METHOD FB_init : BOOL
VAR_INPUT
	bInitRetains : BOOL; // if TRUE, the retain variables are initialized (warm start / cold start)
	bInCopyCode : BOOL;  // if TRUE, the instance afterwards gets moved into the copy code (online change)
END_VAR
AddInput('aElement', aElement);
AddInput('ipContainer', ipContainer);
AddInput('nIndex', nIndex);
AddInput('hrPrev', hrPrev);
AddOutput('ipContainer', ipContainer);
AddOutput('hresult',hresult);
END_METHOD

METHOD PUBLIC  Clone : I_Node
VAR
	pNode : POINTER TO Node_F_VN_SetAt_TcVnVector4_INT;
END_VAR
pNode := __NEW(Node_F_VN_SetAt_TcVnVector4_INT);
Clone := pNode^;
END_METHOD

METHOD PROTECTED OnExecute : HRESULT
hresult.Value := F_VN_SetAt_TcVnVector4_INT(
    aElement := aElement.Value,
    ipContainer := ipContainer.Value,
    nIndex := nIndex.Value,
    hrPrev:= hrPrev.Value);
END_METHOD

METHOD PUBLIC PreExecutionCheck
VAR_INPUT
	Check : I_PreExecutionChecks;
END_VAR
Check.IsTrue(ipContainer.IsValid, 'ipContainer must be a valid container');
END_METHOD

END_FUNCTION_BLOCK

// Nodes/Basic Container Operations/Node_F_VN_SetAt_TcVnVector4_LREAL
{attribute 'linkalways'} 
{attribute 'no_explicit_call' := 'This FB is a CLASS and must be accessed using methods or properties'}
{attribute 'enable_dynamic_creation'}
FUNCTION_BLOCK Node_F_VN_SetAt_TcVnVector4_LREAL EXTENDS VisionNode
VAR
    aElement : _TcVnVector4_LREAL;
    ipContainer : _ITcVnContainer;
    nIndex : _ULINT(0);
    hrPrev : _HRESULT(S_OK);
    hresult : _HRESULT(S_OK);
END_VAR

METHOD FB_init : BOOL
VAR_INPUT
	bInitRetains : BOOL; // if TRUE, the retain variables are initialized (warm start / cold start)
	bInCopyCode : BOOL;  // if TRUE, the instance afterwards gets moved into the copy code (online change)
END_VAR
AddInput('aElement', aElement);
AddInput('ipContainer', ipContainer);
AddInput('nIndex', nIndex);
AddInput('hrPrev', hrPrev);
AddOutput('ipContainer', ipContainer);
AddOutput('hresult',hresult);
END_METHOD

METHOD PUBLIC  Clone : I_Node
VAR
	pNode : POINTER TO Node_F_VN_SetAt_TcVnVector4_LREAL;
END_VAR
pNode := __NEW(Node_F_VN_SetAt_TcVnVector4_LREAL);
Clone := pNode^;
END_METHOD

METHOD PROTECTED OnExecute : HRESULT
hresult.Value := F_VN_SetAt_TcVnVector4_LREAL(
    aElement := aElement.Value,
    ipContainer := ipContainer.Value,
    nIndex := nIndex.Value,
    hrPrev:= hrPrev.Value);
END_METHOD

METHOD PUBLIC PreExecutionCheck
VAR_INPUT
	Check : I_PreExecutionChecks;
END_VAR
Check.IsTrue(ipContainer.IsValid, 'ipContainer must be a valid container');
END_METHOD

END_FUNCTION_BLOCK

// Nodes/Basic Container Operations/Node_F_VN_SetAt_TcVnVector4_SINT
{attribute 'linkalways'} 
{attribute 'no_explicit_call' := 'This FB is a CLASS and must be accessed using methods or properties'}
{attribute 'enable_dynamic_creation'}
FUNCTION_BLOCK Node_F_VN_SetAt_TcVnVector4_SINT EXTENDS VisionNode
VAR
    aElement : _TcVnVector4_SINT;
    ipContainer : _ITcVnContainer;
    nIndex : _ULINT(0);
    hrPrev : _HRESULT(S_OK);
    hresult : _HRESULT(S_OK);
END_VAR

METHOD FB_init : BOOL
VAR_INPUT
	bInitRetains : BOOL; // if TRUE, the retain variables are initialized (warm start / cold start)
	bInCopyCode : BOOL;  // if TRUE, the instance afterwards gets moved into the copy code (online change)
END_VAR
AddInput('aElement', aElement);
AddInput('ipContainer', ipContainer);
AddInput('nIndex', nIndex);
AddInput('hrPrev', hrPrev);
AddOutput('ipContainer', ipContainer);
AddOutput('hresult',hresult);
END_METHOD

METHOD PUBLIC  Clone : I_Node
VAR
	pNode : POINTER TO Node_F_VN_SetAt_TcVnVector4_SINT;
END_VAR
pNode := __NEW(Node_F_VN_SetAt_TcVnVector4_SINT);
Clone := pNode^;
END_METHOD

METHOD PROTECTED OnExecute : HRESULT
hresult.Value := F_VN_SetAt_TcVnVector4_SINT(
    aElement := aElement.Value,
    ipContainer := ipContainer.Value,
    nIndex := nIndex.Value,
    hrPrev:= hrPrev.Value);
END_METHOD

METHOD PUBLIC PreExecutionCheck
VAR_INPUT
	Check : I_PreExecutionChecks;
END_VAR
Check.IsTrue(ipContainer.IsValid, 'ipContainer must be a valid container');
END_METHOD

END_FUNCTION_BLOCK

// Nodes/Basic Container Operations/Node_F_VN_SetAt_TcVnVector4_UINT
{attribute 'linkalways'} 
{attribute 'no_explicit_call' := 'This FB is a CLASS and must be accessed using methods or properties'}
{attribute 'enable_dynamic_creation'}
FUNCTION_BLOCK Node_F_VN_SetAt_TcVnVector4_UINT EXTENDS VisionNode
VAR
    aElement : _TcVnVector4_UINT;
    ipContainer : _ITcVnContainer;
    nIndex : _ULINT(0);
    hrPrev : _HRESULT(S_OK);
    hresult : _HRESULT(S_OK);
END_VAR

METHOD FB_init : BOOL
VAR_INPUT
	bInitRetains : BOOL; // if TRUE, the retain variables are initialized (warm start / cold start)
	bInCopyCode : BOOL;  // if TRUE, the instance afterwards gets moved into the copy code (online change)
END_VAR
AddInput('aElement', aElement);
AddInput('ipContainer', ipContainer);
AddInput('nIndex', nIndex);
AddInput('hrPrev', hrPrev);
AddOutput('ipContainer', ipContainer);
AddOutput('hresult',hresult);
END_METHOD

METHOD PUBLIC  Clone : I_Node
VAR
	pNode : POINTER TO Node_F_VN_SetAt_TcVnVector4_UINT;
END_VAR
pNode := __NEW(Node_F_VN_SetAt_TcVnVector4_UINT);
Clone := pNode^;
END_METHOD

METHOD PROTECTED OnExecute : HRESULT
hresult.Value := F_VN_SetAt_TcVnVector4_UINT(
    aElement := aElement.Value,
    ipContainer := ipContainer.Value,
    nIndex := nIndex.Value,
    hrPrev:= hrPrev.Value);
END_METHOD

METHOD PUBLIC PreExecutionCheck
VAR_INPUT
	Check : I_PreExecutionChecks;
END_VAR
Check.IsTrue(ipContainer.IsValid, 'ipContainer must be a valid container');
END_METHOD

END_FUNCTION_BLOCK

// Nodes/Basic Container Operations/Node_F_VN_SetAt_TcVnVector4_USINT
{attribute 'linkalways'} 
{attribute 'no_explicit_call' := 'This FB is a CLASS and must be accessed using methods or properties'}
{attribute 'enable_dynamic_creation'}
FUNCTION_BLOCK Node_F_VN_SetAt_TcVnVector4_USINT EXTENDS VisionNode
VAR
    aElement : _TcVnVector4_USINT;
    ipContainer : _ITcVnContainer;
    nIndex : _ULINT(0);
    hrPrev : _HRESULT(S_OK);
    hresult : _HRESULT(S_OK);
END_VAR

METHOD FB_init : BOOL
VAR_INPUT
	bInitRetains : BOOL; // if TRUE, the retain variables are initialized (warm start / cold start)
	bInCopyCode : BOOL;  // if TRUE, the instance afterwards gets moved into the copy code (online change)
END_VAR
AddInput('aElement', aElement);
AddInput('ipContainer', ipContainer);
AddInput('nIndex', nIndex);
AddInput('hrPrev', hrPrev);
AddOutput('ipContainer', ipContainer);
AddOutput('hresult',hresult);
END_METHOD

METHOD PUBLIC  Clone : I_Node
VAR
	pNode : POINTER TO Node_F_VN_SetAt_TcVnVector4_USINT;
END_VAR
pNode := __NEW(Node_F_VN_SetAt_TcVnVector4_USINT);
Clone := pNode^;
END_METHOD

METHOD PROTECTED OnExecute : HRESULT
hresult.Value := F_VN_SetAt_TcVnVector4_USINT(
    aElement := aElement.Value,
    ipContainer := ipContainer.Value,
    nIndex := nIndex.Value,
    hrPrev:= hrPrev.Value);
END_METHOD

METHOD PUBLIC PreExecutionCheck
VAR_INPUT
	Check : I_PreExecutionChecks;
END_VAR
Check.IsTrue(ipContainer.IsValid, 'ipContainer must be a valid container');
END_METHOD

END_FUNCTION_BLOCK

// Nodes/Basic Container Operations/Node_F_VN_SetAt_UDINT
{attribute 'linkalways'} 
{attribute 'no_explicit_call' := 'This FB is a CLASS and must be accessed using methods or properties'}
{attribute 'enable_dynamic_creation'}
FUNCTION_BLOCK Node_F_VN_SetAt_UDINT EXTENDS VisionNode
VAR
    nElement : _UDINT(0);
    ipContainer : _ITcVnContainer;
    nIndex : _ULINT(0);
    hrPrev : _HRESULT(S_OK);
    hresult : _HRESULT(S_OK);
END_VAR

METHOD FB_init : BOOL
VAR_INPUT
	bInitRetains : BOOL; // if TRUE, the retain variables are initialized (warm start / cold start)
	bInCopyCode : BOOL;  // if TRUE, the instance afterwards gets moved into the copy code (online change)
END_VAR
AddInput('nElement', nElement);
AddInput('ipContainer', ipContainer);
AddInput('nIndex', nIndex);
AddInput('hrPrev', hrPrev);
AddOutput('ipContainer', ipContainer);
AddOutput('hresult',hresult);
END_METHOD

METHOD PUBLIC  Clone : I_Node
VAR
	pNode : POINTER TO Node_F_VN_SetAt_UDINT;
END_VAR
pNode := __NEW(Node_F_VN_SetAt_UDINT);
Clone := pNode^;
END_METHOD

METHOD PROTECTED OnExecute : HRESULT
hresult.Value := F_VN_SetAt_UDINT(
    nElement := nElement.Value,
    ipContainer := ipContainer.Value,
    nIndex := nIndex.Value,
    hrPrev:= hrPrev.Value);
END_METHOD

METHOD PUBLIC PreExecutionCheck
VAR_INPUT
	Check : I_PreExecutionChecks;
END_VAR
Check.IsTrue(ipContainer.IsValid, 'ipContainer must be a valid container');
Check.IsTrue(ipContainer.HasType('CTcVnContainer_Vector_UDINT'), 'ipContainer contains incorrect types');
END_METHOD

END_FUNCTION_BLOCK

// Nodes/Basic Container Operations/Node_F_VN_SetAt_UINT
{attribute 'linkalways'} 
{attribute 'no_explicit_call' := 'This FB is a CLASS and must be accessed using methods or properties'}
{attribute 'enable_dynamic_creation'}
FUNCTION_BLOCK Node_F_VN_SetAt_UINT EXTENDS VisionNode
VAR
    nElement : _UINT(0);
    ipContainer : _ITcVnContainer;
    nIndex : _ULINT(0);
    hrPrev : _HRESULT(S_OK);
    hresult : _HRESULT(S_OK);
END_VAR

METHOD FB_init : BOOL
VAR_INPUT
	bInitRetains : BOOL; // if TRUE, the retain variables are initialized (warm start / cold start)
	bInCopyCode : BOOL;  // if TRUE, the instance afterwards gets moved into the copy code (online change)
END_VAR
AddInput('nElement', nElement);
AddInput('ipContainer', ipContainer);
AddInput('nIndex', nIndex);
AddInput('hrPrev', hrPrev);
AddOutput('ipContainer', ipContainer);
AddOutput('hresult',hresult);
END_METHOD

METHOD PUBLIC  Clone : I_Node
VAR
	pNode : POINTER TO Node_F_VN_SetAt_UINT;
END_VAR
pNode := __NEW(Node_F_VN_SetAt_UINT);
Clone := pNode^;
END_METHOD

METHOD PROTECTED OnExecute : HRESULT
hresult.Value := F_VN_SetAt_UINT(
    nElement := nElement.Value,
    ipContainer := ipContainer.Value,
    nIndex := nIndex.Value,
    hrPrev:= hrPrev.Value);
END_METHOD

METHOD PUBLIC PreExecutionCheck
VAR_INPUT
	Check : I_PreExecutionChecks;
END_VAR
Check.IsTrue(ipContainer.IsValid, 'ipContainer must be a valid container');
Check.IsTrue(ipContainer.HasType('CTcVnContainer_Vector_UINT'), 'ipContainer contains incorrect types');
END_METHOD

END_FUNCTION_BLOCK

// Nodes/Basic Container Operations/Node_F_VN_SetAt_ULINT
{attribute 'linkalways'} 
{attribute 'no_explicit_call' := 'This FB is a CLASS and must be accessed using methods or properties'}
{attribute 'enable_dynamic_creation'}
FUNCTION_BLOCK Node_F_VN_SetAt_ULINT EXTENDS VisionNode
VAR
    nElement : _ULINT(0);
    ipContainer : _ITcVnContainer;
    nIndex : _ULINT(0);
    hrPrev : _HRESULT(S_OK);
    hresult : _HRESULT(S_OK);
END_VAR

METHOD FB_init : BOOL
VAR_INPUT
	bInitRetains : BOOL; // if TRUE, the retain variables are initialized (warm start / cold start)
	bInCopyCode : BOOL;  // if TRUE, the instance afterwards gets moved into the copy code (online change)
END_VAR
AddInput('nElement', nElement);
AddInput('ipContainer', ipContainer);
AddInput('nIndex', nIndex);
AddInput('hrPrev', hrPrev);
AddOutput('ipContainer', ipContainer);
AddOutput('hresult',hresult);
END_METHOD

METHOD PUBLIC  Clone : I_Node
VAR
	pNode : POINTER TO Node_F_VN_SetAt_ULINT;
END_VAR
pNode := __NEW(Node_F_VN_SetAt_ULINT);
Clone := pNode^;
END_METHOD

METHOD PROTECTED OnExecute : HRESULT
hresult.Value := F_VN_SetAt_ULINT(
    nElement := nElement.Value,
    ipContainer := ipContainer.Value,
    nIndex := nIndex.Value,
    hrPrev:= hrPrev.Value);
END_METHOD

METHOD PUBLIC PreExecutionCheck
VAR_INPUT
	Check : I_PreExecutionChecks;
END_VAR
Check.IsTrue(ipContainer.IsValid, 'ipContainer must be a valid container');
Check.IsTrue(ipContainer.HasType('CTcVnContainer_Vector_ULINT'), 'ipContainer contains incorrect types');
END_METHOD

END_FUNCTION_BLOCK

// Nodes/Basic Container Operations/Node_F_VN_SetAt_USINT
{attribute 'linkalways'} 
{attribute 'no_explicit_call' := 'This FB is a CLASS and must be accessed using methods or properties'}
{attribute 'enable_dynamic_creation'}
FUNCTION_BLOCK Node_F_VN_SetAt_USINT EXTENDS VisionNode
VAR
    nElement : _USINT(0);
    ipContainer : _ITcVnContainer;
    nIndex : _ULINT(0);
    hrPrev : _HRESULT(S_OK);
    hresult : _HRESULT(S_OK);
END_VAR

METHOD FB_init : BOOL
VAR_INPUT
	bInitRetains : BOOL; // if TRUE, the retain variables are initialized (warm start / cold start)
	bInCopyCode : BOOL;  // if TRUE, the instance afterwards gets moved into the copy code (online change)
END_VAR
AddInput('nElement', nElement);
AddInput('ipContainer', ipContainer);
AddInput('nIndex', nIndex);
AddInput('hrPrev', hrPrev);
AddOutput('ipContainer', ipContainer);
AddOutput('hresult',hresult);
END_METHOD

METHOD PUBLIC  Clone : I_Node
VAR
	pNode : POINTER TO Node_F_VN_SetAt_USINT;
END_VAR
pNode := __NEW(Node_F_VN_SetAt_USINT);
Clone := pNode^;
END_METHOD

METHOD PROTECTED OnExecute : HRESULT
hresult.Value := F_VN_SetAt_USINT(
    nElement := nElement.Value,
    ipContainer := ipContainer.Value,
    nIndex := nIndex.Value,
    hrPrev:= hrPrev.Value);
END_METHOD

METHOD PUBLIC PreExecutionCheck
VAR_INPUT
	Check : I_PreExecutionChecks;
END_VAR
Check.IsTrue(ipContainer.IsValid, 'ipContainer must be a valid container');
Check.IsTrue(ipContainer.HasType('CTcVnContainer_Vector_USINT'), 'ipContainer contains incorrect types');
END_METHOD

END_FUNCTION_BLOCK

// Nodes/Basic Image Operations/Node_F_VN_CopyImage
{attribute 'linkalways'} 
{attribute 'no_explicit_call' := 'This FB is a CLASS and must be accessed using methods or properties'}
{attribute 'enable_dynamic_creation'}
FUNCTION_BLOCK Node_F_VN_CopyImage EXTENDS VisionNode
VAR
    ipSrcImage : _ITcVnImage;
    ipDestImage : _ITcVnImage;
    hrPrev : _HRESULT(S_OK);
	hresult : _HRESULT(S_OK);
END_VAR

METHOD FB_init : BOOL
VAR_INPUT
	bInitRetains : BOOL; // if TRUE, the retain variables are initialized (warm start / cold start)
	bInCopyCode : BOOL;  // if TRUE, the instance afterwards gets moved into the copy code (online change)
END_VAR
AddInput('ipSrcImage', ipSrcImage);
AddInput('hrPrev', hrPrev);
AddOutput('ipDestImage', ipDestImage);
AddOutput('hresult',hresult);
END_METHOD

METHOD PUBLIC  Clone : I_Node
VAR
	pNode : POINTER TO Node_F_VN_CopyImage;
END_VAR
pNode := __NEW(Node_F_VN_CopyImage);
Clone := pNode^;
END_METHOD

METHOD PROTECTED OnExecute : HRESULT
hresult.Value := F_VN_CopyImage(
    ipSrcImage := ipSrcImage.Value,
	ipDestImage := ipDestImage.Value,
	hrPrev:= hrPrev.Value);
END_METHOD

METHOD PUBLIC PreExecutionCheck
VAR_INPUT
	Check : I_PreExecutionChecks;
END_VAR
Check.IsTrue(ipSrcImage.IsValid, 'ipSrcImage must contain an image');
END_METHOD

END_FUNCTION_BLOCK

// Nodes/Basic Image Operations/Node_F_VN_GetImageChannel
{attribute 'linkalways'} 
{attribute 'no_explicit_call' := 'This FB is a CLASS and must be accessed using methods or properties'}
{attribute 'enable_dynamic_creation'}
FUNCTION_BLOCK Node_F_VN_GetImageChannel EXTENDS VisionNode
VAR
    ipSrcImage : _ITcVnImage;
    ipDestImage : _ITcVnImage;
    nChannelIndex : _UINT(0);
    hrPrev : _HRESULT(S_OK);
	hresult : _HRESULT(S_OK);
END_VAR

METHOD FB_init : BOOL
VAR_INPUT
	bInitRetains : BOOL; // if TRUE, the retain variables are initialized (warm start / cold start)
	bInCopyCode : BOOL;  // if TRUE, the instance afterwards gets moved into the copy code (online change)
END_VAR
AddInput('ipSrcImage', ipSrcImage);
AddInput('hrPrev', hrPrev);
AddOutput('ipDestImage', ipDestImage);
AddOutput('hresult',hresult);
AddParameter('nChannelIndex', nChannelIndex);
END_METHOD

METHOD PUBLIC  Clone : I_Node
VAR
	pNode : POINTER TO Node_F_VN_GetImageChannel;
END_VAR
pNode := __NEW(Node_F_VN_GetImageChannel);
Clone := pNode^;
END_METHOD

METHOD PROTECTED OnExecute : HRESULT
hresult.Value := F_VN_GetImageChannel(
    ipSrcImage := ipSrcImage.Value,
	ipDestImage := ipDestImage.Value,
    nChannelIndex := nChannelIndex.Value,
	hrPrev:= hrPrev.Value);
END_METHOD

METHOD PUBLIC PreExecutionCheck
VAR_INPUT
	Check : I_PreExecutionChecks;
END_VAR
Check.IsTrue(ipSrcImage.IsValid, 'ipSrcImage must contain an image');
END_METHOD

END_FUNCTION_BLOCK

// Nodes/Basic Image Operations/Node_F_VN_GetImageHeight
{attribute 'linkalways'} 
{attribute 'no_explicit_call' := 'This FB is a CLASS and must be accessed using methods or properties'}
{attribute 'enable_dynamic_creation'}
FUNCTION_BLOCK Node_F_VN_GetImageHeight EXTENDS VisionNode
VAR
    ipImage : _ITcVnImage;
    nHeight : _UDINT(0);
    hrPrev : _HRESULT(S_OK);
	hresult : _HRESULT(S_OK);
END_VAR

METHOD FB_init : BOOL
VAR_INPUT
	bInitRetains : BOOL; // if TRUE, the retain variables are initialized (warm start / cold start)
	bInCopyCode : BOOL;  // if TRUE, the instance afterwards gets moved into the copy code (online change)
END_VAR
AddInput('ipImage', ipImage);
AddInput('hrPrev', hrPrev);
AddOutput('nHeight', nHeight);
AddOutput('hresult', hresult);
END_METHOD

METHOD PUBLIC  Clone : I_Node
VAR
	pNode : POINTER TO Node_F_VN_GetImageHeight;
END_VAR
pNode := __NEW(Node_F_VN_GetImageHeight);
Clone := pNode^;
END_METHOD

METHOD PROTECTED OnExecute : HRESULT
hresult.Value := F_VN_GetImageHeight(
    ipImage := ipImage.Value,
    nHeight := nHeight.Value,
	hrPrev:= hrPrev.Value);
END_METHOD

METHOD PUBLIC PreExecutionCheck
VAR_INPUT
	Check : I_PreExecutionChecks;
END_VAR
Check.IsTrue(ipImage.IsValid, 'ipImage must contain an image');
END_METHOD

END_FUNCTION_BLOCK

// Nodes/Basic Image Operations/Node_F_VN_GetImageInfo
{attribute 'linkalways'} 
{attribute 'no_explicit_call' := 'This FB is a CLASS and must be accessed using methods or properties'}
{attribute 'enable_dynamic_creation'}
FUNCTION_BLOCK Node_F_VN_GetImageInfo EXTENDS VisionNode
VAR
    ipImage : _ITcVnImage;
    stImageInfo : _TcVnImageInfo;
    hrPrev : _HRESULT(S_OK);
	hresult : _HRESULT(S_OK);
END_VAR

METHOD FB_init : BOOL
VAR_INPUT
	bInitRetains : BOOL; // if TRUE, the retain variables are initialized (warm start / cold start)
	bInCopyCode : BOOL;  // if TRUE, the instance afterwards gets moved into the copy code (online change)
END_VAR
AddInput('ipImage', ipImage);
AddInput('hrPrev', hrPrev);
AddOutput('stImageInfo', stImageInfo);
AddOutput('hresult',hresult);
END_METHOD

METHOD PUBLIC  Clone : I_Node
VAR
	pNode : POINTER TO Node_F_VN_GetImageInfo;
END_VAR
pNode := __NEW(Node_F_VN_GetImageInfo);
Clone := pNode^;
END_METHOD

METHOD PROTECTED OnExecute : HRESULT
hresult.Value := F_VN_GetImageInfo(
    ipImage := ipImage.Value,
	stImageInfo := stImageInfo.Value,
	hrPrev:= hrPrev.Value);
END_METHOD

METHOD PUBLIC PreExecutionCheck
VAR_INPUT
	Check : I_PreExecutionChecks;
END_VAR
Check.IsTrue(ipImage.IsValid, 'ipImage must contain an image');
END_METHOD

END_FUNCTION_BLOCK

// Nodes/Basic Image Operations/Node_F_VN_GetImageWidth
{attribute 'linkalways'} 
{attribute 'no_explicit_call' := 'This FB is a CLASS and must be accessed using methods or properties'}
{attribute 'enable_dynamic_creation'}
FUNCTION_BLOCK Node_F_VN_GetImageWidth EXTENDS VisionNode
VAR
    ipImage : _ITcVnImage;
    nWidth : _UDINT(0);
    hrPrev : _HRESULT(S_OK);
	hresult : _HRESULT(S_OK);
END_VAR

METHOD FB_init : BOOL
VAR_INPUT
	bInitRetains : BOOL; // if TRUE, the retain variables are initialized (warm start / cold start)
	bInCopyCode : BOOL;  // if TRUE, the instance afterwards gets moved into the copy code (online change)
END_VAR
AddInput('ipImage', ipImage);
AddInput('hrPrev', hrPrev);
AddOutput('nWidth', nWidth);
AddOutput('hresult',hresult);
END_METHOD

METHOD PUBLIC  Clone : I_Node
VAR
	pNode : POINTER TO Node_F_VN_GetImageWidth;
END_VAR
pNode := __NEW(Node_F_VN_GetImageWidth);
Clone := pNode^;
END_METHOD

METHOD PROTECTED OnExecute : HRESULT
hresult.Value := F_VN_GetImageWidth(
    ipImage := ipImage.Value,
    nWidth := nWidth.Value,
	hrPrev:= hrPrev.Value);
END_METHOD

METHOD PUBLIC PreExecutionCheck
VAR_INPUT
	Check : I_PreExecutionChecks;
END_VAR
Check.IsTrue(ipImage.IsValid, 'ipImage must contain an image');
END_METHOD

END_FUNCTION_BLOCK

// Nodes/Basic Image Operations/Node_F_VN_GetPixelFormat
{attribute 'linkalways'} 
{attribute 'no_explicit_call' := 'This FB is a CLASS and must be accessed using methods or properties'}
{attribute 'enable_dynamic_creation'}
FUNCTION_BLOCK Node_F_VN_GetPixelFormat EXTENDS VisionNode
VAR
    ipImage : _ITcVnImage;
    stPixelFormat : _TcVnPixelFormat;
    hrPrev : _HRESULT(S_OK);
	hresult : _HRESULT(S_OK);
END_VAR

METHOD FB_init : BOOL
VAR_INPUT
	bInitRetains : BOOL; // if TRUE, the retain variables are initialized (warm start / cold start)
	bInCopyCode : BOOL;  // if TRUE, the instance afterwards gets moved into the copy code (online change)
END_VAR
AddInput('ipImage', ipImage);
AddInput('hrPrev', hrPrev);
AddOutput('stPixelFormat', stPixelFormat);
AddOutput('hresult',hresult);
END_METHOD

METHOD PUBLIC  Clone : I_Node
VAR
	pNode : POINTER TO Node_F_VN_GetPixelFormat;
END_VAR
pNode := __NEW(Node_F_VN_GetPixelFormat);
Clone := pNode^;
END_METHOD

METHOD PROTECTED OnExecute : HRESULT
hresult.Value := F_VN_GetPixelFormat(
    ipImage := ipImage.Value,
	stPixelFormat := stPixelFormat.Value,
	hrPrev:= hrPrev.Value);
END_METHOD

METHOD PUBLIC PreExecutionCheck
VAR_INPUT
	Check : I_PreExecutionChecks;
END_VAR
Check.IsTrue(ipImage.IsValid, 'ipImage must contain an image');
END_METHOD

END_FUNCTION_BLOCK

// Nodes/Basic Image Operations/Node_F_VN_SetRoi
{attribute 'linkalways'} 
{attribute 'no_explicit_call' := 'This FB is a CLASS and must be accessed using methods or properties'}
{attribute 'enable_dynamic_creation'}
FUNCTION_BLOCK Node_F_VN_SetRoi EXTENDS VisionNode
VAR
    nX : _UDINT(0);
    nY : _UDINT(0);
    nWidth : _UDINT(0);
    nHeight : _UDINT(0);
    ipDestImage : _ITcVnImage;
    hrPrev : _HRESULT(S_OK);
	hresult : _HRESULT(S_OK);
END_VAR

METHOD FB_init : BOOL
VAR_INPUT
	bInitRetains : BOOL; // if TRUE, the retain variables are initialized (warm start / cold start)
	bInCopyCode : BOOL;  // if TRUE, the instance afterwards gets moved into the copy code (online change)
END_VAR
AddParameter('nX', nX);
AddParameter('nY', nY);
AddParameter('nWidth', nWidth);
AddParameter('nHeight', nHeight);
AddInput('ipDestImage', ipDestImage);
AddInput('hrPrev', hrPrev);
AddOutput('ipDestImage', ipDestImage);
AddOutput('hresult',hresult);
END_METHOD

METHOD PUBLIC  Clone : I_Node
VAR
	pNode : POINTER TO Node_F_VN_SetRoi;
END_VAR
pNode := __NEW(Node_F_VN_SetRoi);
Clone := pNode^;
END_METHOD

METHOD PROTECTED  OnExecute : HRESULT
hresult.Value := F_VN_SetRoi(
    nX := nX.Value,
    nY := nY.Value,
    nWidth := nWidth.Value,
	nHeight := nHeight.Value,
	ipDestImage := ipDestImage.Value,
	hrPrev:= hrPrev.Value);
END_METHOD

METHOD PUBLIC PreExecutionCheck
VAR_INPUT
	Check : I_PreExecutionChecks;
END_VAR
Check.IsTrue(ipDestImage.IsValid, 'ipDestImage must contain an image');
END_METHOD

END_FUNCTION_BLOCK

// Nodes/Constants/Node_RGBA_BLACK
{attribute 'linkalways'} 
{attribute 'no_explicit_call' := 'This FB is a CLASS and must be accessed using methods or properties'}
{attribute 'enable_dynamic_creation'}
FUNCTION_BLOCK Node_RGBA_BLACK EXTENDS VisionNode
VAR
    out : _TcVnVector4_LREAL;
END_VAR

METHOD FB_init : BOOL
VAR_INPUT
	bInitRetains : BOOL; // if TRUE, the retain variables are initialized (warm start / cold start)
	bInCopyCode : BOOL;  // if TRUE, the instance afterwards gets moved into the copy code (online change)
END_VAR
AddOutput('out', out);
END_METHOD

METHOD PUBLIC  Clone : I_Node
VAR
	pNode : POINTER TO Node_RGBA_BLACK;
END_VAR
pNode := __NEW(Node_RGBA_BLACK);
Clone := pNode^;
END_METHOD

METHOD PROTECTED OnExecute : HRESULT
out.Value := GVL_COLOURS.RGBA_BLACK;
END_METHOD

METHOD PUBLIC PreExecutionCheck
VAR_INPUT
	Check : I_PreExecutionChecks;
END_VAR
END_METHOD

END_FUNCTION_BLOCK

// Nodes/Constants/Node_RGBA_BLUE
{attribute 'linkalways'} 
{attribute 'no_explicit_call' := 'This FB is a CLASS and must be accessed using methods or properties'}
{attribute 'enable_dynamic_creation'}
FUNCTION_BLOCK Node_RGBA_BLUE EXTENDS VisionNode
VAR
    out : _TcVnVector4_LREAL;
END_VAR

METHOD FB_init : BOOL
VAR_INPUT
	bInitRetains : BOOL; // if TRUE, the retain variables are initialized (warm start / cold start)
	bInCopyCode : BOOL;  // if TRUE, the instance afterwards gets moved into the copy code (online change)
END_VAR
AddOutput('out', out);
END_METHOD

METHOD PUBLIC  Clone : I_Node
VAR
	pNode : POINTER TO Node_RGBA_BLUE;
END_VAR
pNode := __NEW(Node_RGBA_BLUE);
Clone := pNode^;
END_METHOD

METHOD PROTECTED OnExecute : HRESULT
out.Value := GVL_COLOURS.RGBA_BLUE;
END_METHOD

METHOD PUBLIC PreExecutionCheck
VAR_INPUT
	Check : I_PreExecutionChecks;
END_VAR
END_METHOD

END_FUNCTION_BLOCK

// Nodes/Constants/Node_RGBA_CYAN
{attribute 'linkalways'} 
{attribute 'no_explicit_call' := 'This FB is a CLASS and must be accessed using methods or properties'}
{attribute 'enable_dynamic_creation'}
FUNCTION_BLOCK Node_RGBA_CYAN EXTENDS VisionNode
VAR
    out : _TcVnVector4_LREAL;
END_VAR

METHOD FB_init : BOOL
VAR_INPUT
	bInitRetains : BOOL; // if TRUE, the retain variables are initialized (warm start / cold start)
	bInCopyCode : BOOL;  // if TRUE, the instance afterwards gets moved into the copy code (online change)
END_VAR
AddOutput('out', out);
END_METHOD

METHOD PUBLIC  Clone : I_Node
VAR
	pNode : POINTER TO Node_RGBA_CYAN;
END_VAR
pNode := __NEW(Node_RGBA_CYAN);
Clone := pNode^;
END_METHOD

METHOD PROTECTED OnExecute : HRESULT
out.Value := GVL_COLOURS.RGBA_CYAN;
END_METHOD

METHOD PUBLIC PreExecutionCheck
VAR_INPUT
	Check : I_PreExecutionChecks;
END_VAR
END_METHOD

END_FUNCTION_BLOCK

// Nodes/Constants/Node_RGBA_GREEN
{attribute 'linkalways'} 
{attribute 'no_explicit_call' := 'This FB is a CLASS and must be accessed using methods or properties'}
{attribute 'enable_dynamic_creation'}
FUNCTION_BLOCK Node_RGBA_GREEN EXTENDS VisionNode
VAR
    out : _TcVnVector4_LREAL;
END_VAR

METHOD FB_init : BOOL
VAR_INPUT
	bInitRetains : BOOL; // if TRUE, the retain variables are initialized (warm start / cold start)
	bInCopyCode : BOOL;  // if TRUE, the instance afterwards gets moved into the copy code (online change)
END_VAR
AddOutput('out', out);
END_METHOD

METHOD PUBLIC  Clone : I_Node
VAR
	pNode : POINTER TO Node_RGBA_GREEN;
END_VAR
pNode := __NEW(Node_RGBA_GREEN);
Clone := pNode^;
END_METHOD

METHOD PROTECTED OnExecute : HRESULT
out.Value := GVL_COLOURS.RGBA_GREEN;
END_METHOD

METHOD PUBLIC PreExecutionCheck
VAR_INPUT
	Check : I_PreExecutionChecks;
END_VAR
END_METHOD

END_FUNCTION_BLOCK

// Nodes/Constants/Node_RGBA_MAGENTA
{attribute 'linkalways'} 
{attribute 'no_explicit_call' := 'This FB is a CLASS and must be accessed using methods or properties'}
{attribute 'enable_dynamic_creation'}
FUNCTION_BLOCK Node_RGBA_MAGENTA EXTENDS VisionNode
VAR
    out : _TcVnVector4_LREAL;
END_VAR

METHOD FB_init : BOOL
VAR_INPUT
	bInitRetains : BOOL; // if TRUE, the retain variables are initialized (warm start / cold start)
	bInCopyCode : BOOL;  // if TRUE, the instance afterwards gets moved into the copy code (online change)
END_VAR
AddOutput('out', out);
END_METHOD

METHOD PUBLIC  Clone : I_Node
VAR
	pNode : POINTER TO Node_RGBA_MAGENTA;
END_VAR
pNode := __NEW(Node_RGBA_MAGENTA);
Clone := pNode^;
END_METHOD

METHOD PROTECTED OnExecute : HRESULT
out.Value := GVL_COLOURS.RGBA_MAGENTA;
END_METHOD

METHOD PUBLIC PreExecutionCheck
VAR_INPUT
	Check : I_PreExecutionChecks;
END_VAR
END_METHOD

END_FUNCTION_BLOCK

// Nodes/Constants/Node_RGBA_RED
{attribute 'linkalways'} 
{attribute 'no_explicit_call' := 'This FB is a CLASS and must be accessed using methods or properties'}
{attribute 'enable_dynamic_creation'}
FUNCTION_BLOCK Node_RGBA_RED EXTENDS VisionNode
VAR
    out : _TcVnVector4_LREAL;
END_VAR

METHOD FB_init : BOOL
VAR_INPUT
	bInitRetains : BOOL; // if TRUE, the retain variables are initialized (warm start / cold start)
	bInCopyCode : BOOL;  // if TRUE, the instance afterwards gets moved into the copy code (online change)
END_VAR
AddOutput('out', out);
END_METHOD

METHOD PUBLIC  Clone : I_Node
VAR
	pNode : POINTER TO Node_RGBA_RED;
END_VAR
pNode := __NEW(Node_RGBA_RED);
Clone := pNode^;
END_METHOD

METHOD PROTECTED OnExecute : HRESULT
out.Value := GVL_COLOURS.RGBA_RED;
END_METHOD

METHOD PUBLIC PreExecutionCheck
VAR_INPUT
	Check : I_PreExecutionChecks;
END_VAR
END_METHOD

END_FUNCTION_BLOCK

// Nodes/Constants/Node_RGBA_WHITE
{attribute 'linkalways'} 
{attribute 'no_explicit_call' := 'This FB is a CLASS and must be accessed using methods or properties'}
{attribute 'enable_dynamic_creation'}
FUNCTION_BLOCK Node_RGBA_WHITE EXTENDS VisionNode
VAR
    out : _TcVnVector4_LREAL;
END_VAR

METHOD FB_init : BOOL
VAR_INPUT
	bInitRetains : BOOL; // if TRUE, the retain variables are initialized (warm start / cold start)
	bInCopyCode : BOOL;  // if TRUE, the instance afterwards gets moved into the copy code (online change)
END_VAR
AddOutput('out', out);
END_METHOD

METHOD PUBLIC  Clone : I_Node
VAR
	pNode : POINTER TO Node_RGBA_WHITE;
END_VAR
pNode := __NEW(Node_RGBA_WHITE);
Clone := pNode^;
END_METHOD

METHOD PROTECTED OnExecute : HRESULT
out.Value := GVL_COLOURS.RGBA_WHITE;
END_METHOD

METHOD PUBLIC PreExecutionCheck
VAR_INPUT
	Check : I_PreExecutionChecks;
END_VAR
END_METHOD

END_FUNCTION_BLOCK

// Nodes/Constants/Node_RGBA_YELLOW
{attribute 'linkalways'} 
{attribute 'no_explicit_call' := 'This FB is a CLASS and must be accessed using methods or properties'}
{attribute 'enable_dynamic_creation'}
FUNCTION_BLOCK Node_RGBA_YELLOW EXTENDS VisionNode
VAR
    out : _TcVnVector4_LREAL;
END_VAR

METHOD FB_init : BOOL
VAR_INPUT
	bInitRetains : BOOL; // if TRUE, the retain variables are initialized (warm start / cold start)
	bInCopyCode : BOOL;  // if TRUE, the instance afterwards gets moved into the copy code (online change)
END_VAR
AddOutput('out', out);
END_METHOD

METHOD PUBLIC  Clone : I_Node
VAR
	pNode : POINTER TO Node_RGBA_YELLOW;
END_VAR
pNode := __NEW(Node_RGBA_YELLOW);
Clone := pNode^;
END_METHOD

METHOD PROTECTED OnExecute : HRESULT
out.Value := GVL_COLOURS.RGBA_YELLOW;
END_METHOD

METHOD PUBLIC PreExecutionCheck
VAR_INPUT
	Check : I_PreExecutionChecks;
END_VAR
END_METHOD

END_FUNCTION_BLOCK

// Nodes/Container Statistics/Node_F_VN_MaxElementElementwise_DINT
{attribute 'linkalways'} 
{attribute 'no_explicit_call' := 'This FB is a CLASS and must be accessed using methods or properties'}
{attribute 'enable_dynamic_creation'}
FUNCTION_BLOCK Node_F_VN_MaxElementElementwise_DINT EXTENDS VisionNode
VAR
    ipContainer : _ITcVnContainer;
    nMax : _DINT(0);
    hrPrev : _HRESULT(S_OK);
    hresult : _HRESULT(S_OK);
END_VAR

METHOD FB_init : BOOL
VAR_INPUT
	bInitRetains : BOOL; // if TRUE, the retain variables are initialized (warm start / cold start)
	bInCopyCode : BOOL;  // if TRUE, the instance afterwards gets moved into the copy code (online change)
END_VAR
AddInput('ipContainer', ipContainer);
AddInput('nMax', nMax);
AddInput('hrPrev', hrPrev);
AddOutput('ipContainer', ipContainer);
AddOutput('hresult',hresult);
END_METHOD

METHOD PUBLIC  Clone : I_Node
VAR
	pNode : POINTER TO Node_F_VN_MaxElementElementwise_DINT;
END_VAR
pNode := __NEW(Node_F_VN_MaxElementElementwise_DINT);
Clone := pNode^;
END_METHOD

METHOD PROTECTED OnExecute : HRESULT
hresult.Value := F_VN_MaxElementElementwise_DINT(
    ipContainer := ipContainer.Value,
    nMax := nMax.Value,
    hrPrev:= hrPrev.Value);
END_METHOD

METHOD PUBLIC PreExecutionCheck
VAR_INPUT
	Check : I_PreExecutionChecks;
END_VAR
VAR
    name : STRING;
END_VAR
Check.IsTrue(ipContainer.IsValid, 'ipContainer must be a valid container');
Check.IsTrue(ipContainer.HasType('CTcVnContainer_Vector_DINT'), 'ipContainer contains incorrect types');
END_METHOD

END_FUNCTION_BLOCK

// Nodes/Container Statistics/Node_F_VN_MaxElementElementwise_INT
{attribute 'linkalways'} 
{attribute 'no_explicit_call' := 'This FB is a CLASS and must be accessed using methods or properties'}
{attribute 'enable_dynamic_creation'}
FUNCTION_BLOCK Node_F_VN_MaxElementElementwise_INT EXTENDS VisionNode
VAR
    ipContainer : _ITcVnContainer;
    nMax : _INT(0);
    hrPrev : _HRESULT(S_OK);
    hresult : _HRESULT(S_OK);
END_VAR

METHOD FB_init : BOOL
VAR_INPUT
	bInitRetains : BOOL; // if TRUE, the retain variables are initialized (warm start / cold start)
	bInCopyCode : BOOL;  // if TRUE, the instance afterwards gets moved into the copy code (online change)
END_VAR
AddInput('ipContainer', ipContainer);
AddInput('nMax', nMax);
AddInput('hrPrev', hrPrev);
AddOutput('ipContainer', ipContainer);
AddOutput('hresult',hresult);
END_METHOD

METHOD PUBLIC  Clone : I_Node
VAR
	pNode : POINTER TO Node_F_VN_MaxElementElementwise_INT;
END_VAR
pNode := __NEW(Node_F_VN_MaxElementElementwise_INT);
Clone := pNode^;
END_METHOD

METHOD PROTECTED OnExecute : HRESULT
hresult.Value := F_VN_MaxElementElementwise_INT(
    ipContainer := ipContainer.Value,
    nMax := nMax.Value,
    hrPrev:= hrPrev.Value);
END_METHOD

METHOD PUBLIC PreExecutionCheck
VAR_INPUT
	Check : I_PreExecutionChecks;
END_VAR
Check.IsTrue(ipContainer.IsValid, 'ipContainer must be a valid container');
Check.IsTrue(ipContainer.HasType('CTcVnContainer_Vector_INT'), 'ipContainer contains incorrect types');
END_METHOD

END_FUNCTION_BLOCK

// Nodes/Container Statistics/Node_F_VN_MaxElementElementwise_LREAL
{attribute 'linkalways'} 
{attribute 'no_explicit_call' := 'This FB is a CLASS and must be accessed using methods or properties'}
{attribute 'enable_dynamic_creation'}
FUNCTION_BLOCK Node_F_VN_MaxElementElementwise_LREAL EXTENDS VisionNode
VAR
    ipContainer : _ITcVnContainer;
    fMax : _LREAL(0.0);
    hrPrev : _HRESULT(S_OK);
    hresult : _HRESULT(S_OK);
END_VAR

METHOD FB_init : BOOL
VAR_INPUT
	bInitRetains : BOOL; // if TRUE, the retain variables are initialized (warm start / cold start)
	bInCopyCode : BOOL;  // if TRUE, the instance afterwards gets moved into the copy code (online change)
END_VAR
AddInput('ipContainer', ipContainer);
AddInput('fMax', fMax);
AddInput('hrPrev', hrPrev);
AddOutput('ipContainer', ipContainer);
AddOutput('hresult',hresult);
END_METHOD

METHOD PUBLIC  Clone : I_Node
VAR
	pNode : POINTER TO Node_F_VN_MaxElementElementwise_LREAL;
END_VAR
pNode := __NEW(Node_F_VN_MaxElementElementwise_LREAL);
Clone := pNode^;
END_METHOD

METHOD PROTECTED OnExecute : HRESULT
hresult.Value := F_VN_MaxElementElementwise_LREAL(
    ipContainer := ipContainer.Value,
    fMax := fMax.Value,
    hrPrev:= hrPrev.Value);
END_METHOD

METHOD PUBLIC PreExecutionCheck
VAR_INPUT
	Check : I_PreExecutionChecks;
END_VAR
Check.IsTrue(ipContainer.IsValid, 'ipContainer must be a valid container');
Check.IsTrue(ipContainer.HasType('CTcVnContainer_Vector_LREAL'), 'ipContainer contains incorrect types');
END_METHOD

END_FUNCTION_BLOCK

// Nodes/Container Statistics/Node_F_VN_MaxElementElementwise_REAL
{attribute 'linkalways'} 
{attribute 'no_explicit_call' := 'This FB is a CLASS and must be accessed using methods or properties'}
{attribute 'enable_dynamic_creation'}
FUNCTION_BLOCK Node_F_VN_MaxElementElementwise_REAL EXTENDS VisionNode
VAR
    ipContainer : _ITcVnContainer;
    fMax : _REAL(0.0);
    hrPrev : _HRESULT(S_OK);
    hresult : _HRESULT(S_OK);
END_VAR

METHOD FB_init : BOOL
VAR_INPUT
	bInitRetains : BOOL; // if TRUE, the retain variables are initialized (warm start / cold start)
	bInCopyCode : BOOL;  // if TRUE, the instance afterwards gets moved into the copy code (online change)
END_VAR
AddInput('ipContainer', ipContainer);
AddInput('fMax', fMax);
AddInput('hrPrev', hrPrev);
AddOutput('ipContainer', ipContainer);
AddOutput('hresult',hresult);
END_METHOD

METHOD PUBLIC  Clone : I_Node
VAR
	pNode : POINTER TO Node_F_VN_MaxElementElementwise_REAL;
END_VAR
pNode := __NEW(Node_F_VN_MaxElementElementwise_REAL);
Clone := pNode^;
END_METHOD

METHOD PROTECTED OnExecute : HRESULT
hresult.Value := F_VN_MaxElementElementwise_REAL(
    ipContainer := ipContainer.Value,
    fMax := fMax.Value,
    hrPrev:= hrPrev.Value);
END_METHOD

METHOD PUBLIC PreExecutionCheck
VAR_INPUT
	Check : I_PreExecutionChecks;
END_VAR
Check.IsTrue(ipContainer.IsValid, 'ipContainer must be a valid container');
Check.IsTrue(ipContainer.HasType('CTcVnContainer_Vector_REAL'), 'ipContainer contains incorrect types');
END_METHOD

END_FUNCTION_BLOCK

// Nodes/Container Statistics/Node_F_VN_MaxElementElementwise_SINT
{attribute 'linkalways'} 
{attribute 'no_explicit_call' := 'This FB is a CLASS and must be accessed using methods or properties'}
{attribute 'enable_dynamic_creation'}
FUNCTION_BLOCK Node_F_VN_MaxElementElementwise_SINT EXTENDS VisionNode
VAR
    ipContainer : _ITcVnContainer;
    nMax : _SINT(0);
    hrPrev : _HRESULT(S_OK);
    hresult : _HRESULT(S_OK);
END_VAR

METHOD FB_init : BOOL
VAR_INPUT
	bInitRetains : BOOL; // if TRUE, the retain variables are initialized (warm start / cold start)
	bInCopyCode : BOOL;  // if TRUE, the instance afterwards gets moved into the copy code (online change)
END_VAR
AddInput('ipContainer', ipContainer);
AddInput('nMax', nMax);
AddInput('hrPrev', hrPrev);
AddOutput('ipContainer', ipContainer);
AddOutput('hresult',hresult);
END_METHOD

METHOD PUBLIC  Clone : I_Node
VAR
	pNode : POINTER TO Node_F_VN_MaxElementElementwise_SINT;
END_VAR
pNode := __NEW(Node_F_VN_MaxElementElementwise_SINT);
Clone := pNode^;
END_METHOD

METHOD PROTECTED OnExecute : HRESULT
hresult.Value := F_VN_MaxElementElementwise_SINT(
    ipContainer := ipContainer.Value,
    nMax := nMax.Value,
    hrPrev:= hrPrev.Value);
END_METHOD

METHOD PUBLIC PreExecutionCheck
VAR_INPUT
	Check : I_PreExecutionChecks;
END_VAR
Check.IsTrue(ipContainer.IsValid, 'ipContainer must be a valid container');
Check.IsTrue(ipContainer.HasType('CTcVnContainer_Vector_SINT'), 'ipContainer contains incorrect types');
END_METHOD

END_FUNCTION_BLOCK

// Nodes/Container Statistics/Node_F_VN_MaxElementElementwise_TcVnPoint2_DINT
{attribute 'linkalways'} 
{attribute 'no_explicit_call' := 'This FB is a CLASS and must be accessed using methods or properties'}
{attribute 'enable_dynamic_creation'}
FUNCTION_BLOCK Node_F_VN_MaxElementElementwise_TcVnPoint2_DINT EXTENDS VisionNode
VAR
    ipContainer : _ITcVnContainer;
    aMax : _TcVnPoint2_DINT;
    hrPrev : _HRESULT(S_OK);
    hresult : _HRESULT(S_OK);
END_VAR

METHOD FB_init : BOOL
VAR_INPUT
	bInitRetains : BOOL; // if TRUE, the retain variables are initialized (warm start / cold start)
	bInCopyCode : BOOL;  // if TRUE, the instance afterwards gets moved into the copy code (online change)
END_VAR
AddInput('ipContainer', ipContainer);
AddInput('aMax', aMax);
AddInput('hrPrev', hrPrev);
AddOutput('ipContainer', ipContainer);
AddOutput('hresult',hresult);
END_METHOD

METHOD PUBLIC  Clone : I_Node
VAR
	pNode : POINTER TO Node_F_VN_MaxElementElementwise_TcVnPoint2_DINT;
END_VAR
pNode := __NEW(Node_F_VN_MaxElementElementwise_TcVnPoint2_DINT);
Clone := pNode^;
END_METHOD

METHOD PROTECTED OnExecute : HRESULT
hresult.Value := F_VN_MaxElementElementwise_TcVnPoint2_DINT(
    ipContainer := ipContainer.Value,
    aMax := aMax.Value,
    hrPrev:= hrPrev.Value);
END_METHOD

METHOD PUBLIC PreExecutionCheck
VAR_INPUT
	Check : I_PreExecutionChecks;
END_VAR
Check.IsTrue(ipContainer.IsValid, 'ipContainer must be a valid container');
END_METHOD

END_FUNCTION_BLOCK

// Nodes/Container Statistics/Node_F_VN_MaxElementElementwise_TcVnPoint2_LREAL
{attribute 'linkalways'} 
{attribute 'no_explicit_call' := 'This FB is a CLASS and must be accessed using methods or properties'}
{attribute 'enable_dynamic_creation'}
FUNCTION_BLOCK Node_F_VN_MaxElementElementwise_TcVnPoint2_LREAL EXTENDS VisionNode
VAR
    ipContainer : _ITcVnContainer;
    aMax : _TcVnPoint2_LREAL;
    hrPrev : _HRESULT(S_OK);
    hresult : _HRESULT(S_OK);
END_VAR

METHOD FB_init : BOOL
VAR_INPUT
	bInitRetains : BOOL; // if TRUE, the retain variables are initialized (warm start / cold start)
	bInCopyCode : BOOL;  // if TRUE, the instance afterwards gets moved into the copy code (online change)
END_VAR
AddInput('ipContainer', ipContainer);
AddInput('aMax', aMax);
AddInput('hrPrev', hrPrev);
AddOutput('ipContainer', ipContainer);
AddOutput('hresult',hresult);
END_METHOD

METHOD PUBLIC  Clone : I_Node
VAR
	pNode : POINTER TO Node_F_VN_MaxElementElementwise_TcVnPoint2_LREAL;
END_VAR
pNode := __NEW(Node_F_VN_MaxElementElementwise_TcVnPoint2_LREAL);
Clone := pNode^;
END_METHOD

METHOD PROTECTED OnExecute : HRESULT
hresult.Value := F_VN_MaxElementElementwise_TcVnPoint2_LREAL(
    ipContainer := ipContainer.Value,
    aMax := aMax.Value,
    hrPrev:= hrPrev.Value);
END_METHOD

METHOD PUBLIC PreExecutionCheck
VAR_INPUT
	Check : I_PreExecutionChecks;
END_VAR
Check.IsTrue(ipContainer.IsValid, 'ipContainer must be a valid container');
END_METHOD

END_FUNCTION_BLOCK

// Nodes/Container Statistics/Node_F_VN_MaxElementElementwise_TcVnPoint2_REAL
{attribute 'linkalways'} 
{attribute 'no_explicit_call' := 'This FB is a CLASS and must be accessed using methods or properties'}
{attribute 'enable_dynamic_creation'}
FUNCTION_BLOCK Node_F_VN_MaxElementElementwise_TcVnPoint2_REAL EXTENDS VisionNode
VAR
    ipContainer : _ITcVnContainer;
    aMax : _TcVnPoint2_REAL;
    hrPrev : _HRESULT(S_OK);
    hresult : _HRESULT(S_OK);
END_VAR

METHOD FB_init : BOOL
VAR_INPUT
	bInitRetains : BOOL; // if TRUE, the retain variables are initialized (warm start / cold start)
	bInCopyCode : BOOL;  // if TRUE, the instance afterwards gets moved into the copy code (online change)
END_VAR
AddInput('ipContainer', ipContainer);
AddInput('aMax', aMax);
AddInput('hrPrev', hrPrev);
AddOutput('ipContainer', ipContainer);
AddOutput('hresult',hresult);
END_METHOD

METHOD PUBLIC  Clone : I_Node
VAR
	pNode : POINTER TO Node_F_VN_MaxElementElementwise_TcVnPoint2_REAL;
END_VAR
pNode := __NEW(Node_F_VN_MaxElementElementwise_TcVnPoint2_REAL);
Clone := pNode^;
END_METHOD

METHOD PROTECTED OnExecute : HRESULT
hresult.Value := F_VN_MaxElementElementwise_TcVnPoint2_REAL(
    ipContainer := ipContainer.Value,
    aMax := aMax.Value,
    hrPrev:= hrPrev.Value);
END_METHOD

METHOD PUBLIC PreExecutionCheck
VAR_INPUT
	Check : I_PreExecutionChecks;
END_VAR
Check.IsTrue(ipContainer.IsValid, 'ipContainer must be a valid container');
END_METHOD

END_FUNCTION_BLOCK

// Nodes/Container Statistics/Node_F_VN_MaxElementElementwise_TcVnPoint3_LREAL
{attribute 'linkalways'} 
{attribute 'no_explicit_call' := 'This FB is a CLASS and must be accessed using methods or properties'}
{attribute 'enable_dynamic_creation'}
FUNCTION_BLOCK Node_F_VN_MaxElementElementwise_TcVnPoint3_LREAL EXTENDS VisionNode
VAR
    ipContainer : _ITcVnContainer;
    aMax : _TcVnPoint3_LREAL;
    hrPrev : _HRESULT(S_OK);
    hresult : _HRESULT(S_OK);
END_VAR

METHOD FB_init : BOOL
VAR_INPUT
	bInitRetains : BOOL; // if TRUE, the retain variables are initialized (warm start / cold start)
	bInCopyCode : BOOL;  // if TRUE, the instance afterwards gets moved into the copy code (online change)
END_VAR
AddInput('ipContainer', ipContainer);
AddInput('aMax', aMax);
AddInput('hrPrev', hrPrev);
AddOutput('ipContainer', ipContainer);
AddOutput('hresult',hresult);
END_METHOD

METHOD PUBLIC  Clone : I_Node
VAR
	pNode : POINTER TO Node_F_VN_MaxElementElementwise_TcVnPoint3_LREAL;
END_VAR
pNode := __NEW(Node_F_VN_MaxElementElementwise_TcVnPoint3_LREAL);
Clone := pNode^;
END_METHOD

METHOD PROTECTED OnExecute : HRESULT
hresult.Value := F_VN_MaxElementElementwise_TcVnPoint3_LREAL(
    ipContainer := ipContainer.Value,
    aMax := aMax.Value,
    hrPrev:= hrPrev.Value);
END_METHOD

METHOD PUBLIC PreExecutionCheck
VAR_INPUT
	Check : I_PreExecutionChecks;
END_VAR
Check.IsTrue(ipContainer.IsValid, 'ipContainer must be a valid container');
END_METHOD

END_FUNCTION_BLOCK

// Nodes/Container Statistics/Node_F_VN_MaxElementElementwise_TcVnPoint3_REAL
{attribute 'linkalways'} 
{attribute 'no_explicit_call' := 'This FB is a CLASS and must be accessed using methods or properties'}
{attribute 'enable_dynamic_creation'}
FUNCTION_BLOCK Node_F_VN_MaxElementElementwise_TcVnPoint3_REAL EXTENDS VisionNode
VAR
    ipContainer : _ITcVnContainer;
    aMax : _TcVnPoint3_REAL;
    hrPrev : _HRESULT(S_OK);
    hresult : _HRESULT(S_OK);
END_VAR

METHOD FB_init : BOOL
VAR_INPUT
	bInitRetains : BOOL; // if TRUE, the retain variables are initialized (warm start / cold start)
	bInCopyCode : BOOL;  // if TRUE, the instance afterwards gets moved into the copy code (online change)
END_VAR
AddInput('ipContainer', ipContainer);
AddInput('aMax', aMax);
AddInput('hrPrev', hrPrev);
AddOutput('ipContainer', ipContainer);
AddOutput('hresult',hresult);
END_METHOD

METHOD PUBLIC  Clone : I_Node
VAR
	pNode : POINTER TO Node_F_VN_MaxElementElementwise_TcVnPoint3_REAL;
END_VAR
pNode := __NEW(Node_F_VN_MaxElementElementwise_TcVnPoint3_REAL);
Clone := pNode^;
END_METHOD

METHOD PROTECTED OnExecute : HRESULT
hresult.Value := F_VN_MaxElementElementwise_TcVnPoint3_REAL(
    ipContainer := ipContainer.Value,
    aMax := aMax.Value,
    hrPrev:= hrPrev.Value);
END_METHOD

METHOD PUBLIC PreExecutionCheck
VAR_INPUT
	Check : I_PreExecutionChecks;
END_VAR
Check.IsTrue(ipContainer.IsValid, 'ipContainer must be a valid container');
END_METHOD

END_FUNCTION_BLOCK

// Nodes/Container Statistics/Node_F_VN_MaxElementElementwise_TcVnVector2_DINT
{attribute 'linkalways'} 
{attribute 'no_explicit_call' := 'This FB is a CLASS and must be accessed using methods or properties'}
{attribute 'enable_dynamic_creation'}
FUNCTION_BLOCK Node_F_VN_MaxElementElementwise_TcVnVector2_DINT EXTENDS VisionNode
VAR
    ipContainer : _ITcVnContainer;
    aMax : _TcVnVector2_DINT;
    hrPrev : _HRESULT(S_OK);
    hresult : _HRESULT(S_OK);
END_VAR

METHOD FB_init : BOOL
VAR_INPUT
	bInitRetains : BOOL; // if TRUE, the retain variables are initialized (warm start / cold start)
	bInCopyCode : BOOL;  // if TRUE, the instance afterwards gets moved into the copy code (online change)
END_VAR
AddInput('ipContainer', ipContainer);
AddInput('aMax', aMax);
AddInput('hrPrev', hrPrev);
AddOutput('ipContainer', ipContainer);
AddOutput('hresult',hresult);
END_METHOD

METHOD PUBLIC  Clone : I_Node
VAR
	pNode : POINTER TO Node_F_VN_MaxElementElementwise_TcVnVector2_DINT;
END_VAR
pNode := __NEW(Node_F_VN_MaxElementElementwise_TcVnVector2_DINT);
Clone := pNode^;
END_METHOD

METHOD PROTECTED OnExecute : HRESULT
hresult.Value := F_VN_MaxElementElementwise_TcVnVector2_DINT(
    ipContainer := ipContainer.Value,
    aMax := aMax.Value,
    hrPrev:= hrPrev.Value);
END_METHOD

METHOD PUBLIC PreExecutionCheck
VAR_INPUT
	Check : I_PreExecutionChecks;
END_VAR
Check.IsTrue(ipContainer.IsValid, 'ipContainer must be a valid container');
END_METHOD

END_FUNCTION_BLOCK

// Nodes/Container Statistics/Node_F_VN_MaxElementElementwise_TcVnVector2_INT
{attribute 'linkalways'} 
{attribute 'no_explicit_call' := 'This FB is a CLASS and must be accessed using methods or properties'}
{attribute 'enable_dynamic_creation'}
FUNCTION_BLOCK Node_F_VN_MaxElementElementwise_TcVnVector2_INT EXTENDS VisionNode
VAR
    ipContainer : _ITcVnContainer;
    aMax : _TcVnVector2_INT;
    hrPrev : _HRESULT(S_OK);
    hresult : _HRESULT(S_OK);
END_VAR

METHOD FB_init : BOOL
VAR_INPUT
	bInitRetains : BOOL; // if TRUE, the retain variables are initialized (warm start / cold start)
	bInCopyCode : BOOL;  // if TRUE, the instance afterwards gets moved into the copy code (online change)
END_VAR
AddInput('ipContainer', ipContainer);
AddInput('aMax', aMax);
AddInput('hrPrev', hrPrev);
AddOutput('ipContainer', ipContainer);
AddOutput('hresult',hresult);
END_METHOD

METHOD PUBLIC  Clone : I_Node
VAR
	pNode : POINTER TO Node_F_VN_MaxElementElementwise_TcVnVector2_INT;
END_VAR
pNode := __NEW(Node_F_VN_MaxElementElementwise_TcVnVector2_INT);
Clone := pNode^;
END_METHOD

METHOD PROTECTED OnExecute : HRESULT
hresult.Value := F_VN_MaxElementElementwise_TcVnVector2_INT(
    ipContainer := ipContainer.Value,
    aMax := aMax.Value,
    hrPrev:= hrPrev.Value);
END_METHOD

METHOD PUBLIC PreExecutionCheck
VAR_INPUT
	Check : I_PreExecutionChecks;
END_VAR
Check.IsTrue(ipContainer.IsValid, 'ipContainer must be a valid container');
END_METHOD

END_FUNCTION_BLOCK

// Nodes/Container Statistics/Node_F_VN_MaxElementElementwise_TcVnVector2_REAL
{attribute 'linkalways'} 
{attribute 'no_explicit_call' := 'This FB is a CLASS and must be accessed using methods or properties'}
{attribute 'enable_dynamic_creation'}
FUNCTION_BLOCK Node_F_VN_MaxElementElementwise_TcVnVector2_REAL EXTENDS VisionNode
VAR
    ipContainer : _ITcVnContainer;
    aMax : _TcVnVector2_REAL;
    hrPrev : _HRESULT(S_OK);
    hresult : _HRESULT(S_OK);
END_VAR

METHOD FB_init : BOOL
VAR_INPUT
	bInitRetains : BOOL; // if TRUE, the retain variables are initialized (warm start / cold start)
	bInCopyCode : BOOL;  // if TRUE, the instance afterwards gets moved into the copy code (online change)
END_VAR
AddInput('ipContainer', ipContainer);
AddInput('aMax', aMax);
AddInput('hrPrev', hrPrev);
AddOutput('ipContainer', ipContainer);
AddOutput('hresult',hresult);
END_METHOD

METHOD PUBLIC  Clone : I_Node
VAR
	pNode : POINTER TO Node_F_VN_MaxElementElementwise_TcVnVector2_REAL;
END_VAR
pNode := __NEW(Node_F_VN_MaxElementElementwise_TcVnVector2_REAL);
Clone := pNode^;
END_METHOD

METHOD PROTECTED OnExecute : HRESULT
hresult.Value := F_VN_MaxElementElementwise_TcVnVector2_REAL(
    ipContainer := ipContainer.Value,
    aMax := aMax.Value,
    hrPrev:= hrPrev.Value);
END_METHOD

METHOD PUBLIC PreExecutionCheck
VAR_INPUT
	Check : I_PreExecutionChecks;
END_VAR
Check.IsTrue(ipContainer.IsValid, 'ipContainer must be a valid container');
END_METHOD

END_FUNCTION_BLOCK

// Nodes/Container Statistics/Node_F_VN_MaxElementElementwise_TcVnVector2_SINT
{attribute 'linkalways'} 
{attribute 'no_explicit_call' := 'This FB is a CLASS and must be accessed using methods or properties'}
{attribute 'enable_dynamic_creation'}
FUNCTION_BLOCK Node_F_VN_MaxElementElementwise_TcVnVector2_SINT EXTENDS VisionNode
VAR
    ipContainer : _ITcVnContainer;
    aMax : _TcVnVector2_SINT;
    hrPrev : _HRESULT(S_OK);
    hresult : _HRESULT(S_OK);
END_VAR

METHOD FB_init : BOOL
VAR_INPUT
	bInitRetains : BOOL; // if TRUE, the retain variables are initialized (warm start / cold start)
	bInCopyCode : BOOL;  // if TRUE, the instance afterwards gets moved into the copy code (online change)
END_VAR
AddInput('ipContainer', ipContainer);
AddInput('aMax', aMax);
AddInput('hrPrev', hrPrev);
AddOutput('ipContainer', ipContainer);
AddOutput('hresult',hresult);
END_METHOD

METHOD PUBLIC  Clone : I_Node
VAR
	pNode : POINTER TO Node_F_VN_MaxElementElementwise_TcVnVector2_SINT;
END_VAR
pNode := __NEW(Node_F_VN_MaxElementElementwise_TcVnVector2_SINT);
Clone := pNode^;
END_METHOD

METHOD PROTECTED OnExecute : HRESULT
hresult.Value := F_VN_MaxElementElementwise_TcVnVector2_SINT(
    ipContainer := ipContainer.Value,
    aMax := aMax.Value,
    hrPrev:= hrPrev.Value);
END_METHOD

METHOD PUBLIC PreExecutionCheck
VAR_INPUT
	Check : I_PreExecutionChecks;
END_VAR
Check.IsTrue(ipContainer.IsValid, 'ipContainer must be a valid container');
END_METHOD

END_FUNCTION_BLOCK

// Nodes/Container Statistics/Node_F_VN_MaxElementElementwise_TcVnVector2_UINT
{attribute 'linkalways'} 
{attribute 'no_explicit_call' := 'This FB is a CLASS and must be accessed using methods or properties'}
{attribute 'enable_dynamic_creation'}
FUNCTION_BLOCK Node_F_VN_MaxElementElementwise_TcVnVector2_UINT EXTENDS VisionNode
VAR
    ipContainer : _ITcVnContainer;
    aMax : _TcVnVector2_UINT;
    hrPrev : _HRESULT(S_OK);
    hresult : _HRESULT(S_OK);
END_VAR

METHOD FB_init : BOOL
VAR_INPUT
	bInitRetains : BOOL; // if TRUE, the retain variables are initialized (warm start / cold start)
	bInCopyCode : BOOL;  // if TRUE, the instance afterwards gets moved into the copy code (online change)
END_VAR
AddInput('ipContainer', ipContainer);
AddInput('aMax', aMax);
AddInput('hrPrev', hrPrev);
AddOutput('ipContainer', ipContainer);
AddOutput('hresult',hresult);
END_METHOD

METHOD PUBLIC  Clone : I_Node
VAR
	pNode : POINTER TO Node_F_VN_MaxElementElementwise_TcVnVector2_UINT;
END_VAR
pNode := __NEW(Node_F_VN_MaxElementElementwise_TcVnVector2_UINT);
Clone := pNode^;
END_METHOD

METHOD PROTECTED OnExecute : HRESULT
hresult.Value := F_VN_MaxElementElementwise_TcVnVector2_UINT(
    ipContainer := ipContainer.Value,
    aMax := aMax.Value,
    hrPrev:= hrPrev.Value);
END_METHOD

METHOD PUBLIC PreExecutionCheck
VAR_INPUT
	Check : I_PreExecutionChecks;
END_VAR
Check.IsTrue(ipContainer.IsValid, 'ipContainer must be a valid container');
END_METHOD

END_FUNCTION_BLOCK

// Nodes/Container Statistics/Node_F_VN_MaxElementElementwise_TcVnVector2_USINT
{attribute 'linkalways'} 
{attribute 'no_explicit_call' := 'This FB is a CLASS and must be accessed using methods or properties'}
{attribute 'enable_dynamic_creation'}
FUNCTION_BLOCK Node_F_VN_MaxElementElementwise_TcVnVector2_USINT EXTENDS VisionNode
VAR
    ipContainer : _ITcVnContainer;
    aMax : _TcVnVector2_USINT;
    hrPrev : _HRESULT(S_OK);
    hresult : _HRESULT(S_OK);
END_VAR

METHOD FB_init : BOOL
VAR_INPUT
	bInitRetains : BOOL; // if TRUE, the retain variables are initialized (warm start / cold start)
	bInCopyCode : BOOL;  // if TRUE, the instance afterwards gets moved into the copy code (online change)
END_VAR
AddInput('ipContainer', ipContainer);
AddInput('aMax', aMax);
AddInput('hrPrev', hrPrev);
AddOutput('ipContainer', ipContainer);
AddOutput('hresult',hresult);
END_METHOD

METHOD PUBLIC  Clone : I_Node
VAR
	pNode : POINTER TO Node_F_VN_MaxElementElementwise_TcVnVector2_USINT;
END_VAR
pNode := __NEW(Node_F_VN_MaxElementElementwise_TcVnVector2_USINT);
Clone := pNode^;
END_METHOD

METHOD PROTECTED OnExecute : HRESULT
hresult.Value := F_VN_MaxElementElementwise_TcVnVector2_USINT(
    ipContainer := ipContainer.Value,
    aMax := aMax.Value,
    hrPrev:= hrPrev.Value);
END_METHOD

METHOD PUBLIC PreExecutionCheck
VAR_INPUT
	Check : I_PreExecutionChecks;
END_VAR
Check.IsTrue(ipContainer.IsValid, 'ipContainer must be a valid container');
END_METHOD

END_FUNCTION_BLOCK

// Nodes/Container Statistics/Node_F_VN_MaxElementElementwise_TcVnVector3_INT
{attribute 'linkalways'} 
{attribute 'no_explicit_call' := 'This FB is a CLASS and must be accessed using methods or properties'}
{attribute 'enable_dynamic_creation'}
FUNCTION_BLOCK Node_F_VN_MaxElementElementwise_TcVnVector3_INT EXTENDS VisionNode
VAR
    ipContainer : _ITcVnContainer;
    aMax : _TcVnVector3_INT;
    hrPrev : _HRESULT(S_OK);
    hresult : _HRESULT(S_OK);
END_VAR

METHOD FB_init : BOOL
VAR_INPUT
	bInitRetains : BOOL; // if TRUE, the retain variables are initialized (warm start / cold start)
	bInCopyCode : BOOL;  // if TRUE, the instance afterwards gets moved into the copy code (online change)
END_VAR
AddInput('ipContainer', ipContainer);
AddInput('aMax', aMax);
AddInput('hrPrev', hrPrev);
AddOutput('ipContainer', ipContainer);
AddOutput('hresult',hresult);
END_METHOD

METHOD PUBLIC  Clone : I_Node
VAR
	pNode : POINTER TO Node_F_VN_MaxElementElementwise_TcVnVector3_INT;
END_VAR
pNode := __NEW(Node_F_VN_MaxElementElementwise_TcVnVector3_INT);
Clone := pNode^;
END_METHOD

METHOD PROTECTED OnExecute : HRESULT
hresult.Value := F_VN_MaxElementElementwise_TcVnVector3_INT(
    ipContainer := ipContainer.Value,
    aMax := aMax.Value,
    hrPrev:= hrPrev.Value);
END_METHOD

METHOD PUBLIC PreExecutionCheck
VAR_INPUT
	Check : I_PreExecutionChecks;
END_VAR
Check.IsTrue(ipContainer.IsValid, 'ipContainer must be a valid container');
END_METHOD

END_FUNCTION_BLOCK

// Nodes/Container Statistics/Node_F_VN_MaxElementElementwise_TcVnVector3_REAL
{attribute 'linkalways'} 
{attribute 'no_explicit_call' := 'This FB is a CLASS and must be accessed using methods or properties'}
{attribute 'enable_dynamic_creation'}
FUNCTION_BLOCK Node_F_VN_MaxElementElementwise_TcVnVector3_REAL EXTENDS VisionNode
VAR
    ipContainer : _ITcVnContainer;
    aMax : _TcVnVector3_REAL;
    hrPrev : _HRESULT(S_OK);
    hresult : _HRESULT(S_OK);
END_VAR

METHOD FB_init : BOOL
VAR_INPUT
	bInitRetains : BOOL; // if TRUE, the retain variables are initialized (warm start / cold start)
	bInCopyCode : BOOL;  // if TRUE, the instance afterwards gets moved into the copy code (online change)
END_VAR
AddInput('ipContainer', ipContainer);
AddInput('aMax', aMax);
AddInput('hrPrev', hrPrev);
AddOutput('ipContainer', ipContainer);
AddOutput('hresult',hresult);
END_METHOD

METHOD PUBLIC  Clone : I_Node
VAR
	pNode : POINTER TO Node_F_VN_MaxElementElementwise_TcVnVector3_REAL;
END_VAR
pNode := __NEW(Node_F_VN_MaxElementElementwise_TcVnVector3_REAL);
Clone := pNode^;
END_METHOD

METHOD PROTECTED OnExecute : HRESULT
hresult.Value := F_VN_MaxElementElementwise_TcVnVector3_REAL(
    ipContainer := ipContainer.Value,
    aMax := aMax.Value,
    hrPrev:= hrPrev.Value);
END_METHOD

METHOD PUBLIC PreExecutionCheck
VAR_INPUT
	Check : I_PreExecutionChecks;
END_VAR
Check.IsTrue(ipContainer.IsValid, 'ipContainer must be a valid container');
END_METHOD

END_FUNCTION_BLOCK

// Nodes/Container Statistics/Node_F_VN_MaxElementElementwise_TcVnVector3_SINT
{attribute 'linkalways'} 
{attribute 'no_explicit_call' := 'This FB is a CLASS and must be accessed using methods or properties'}
{attribute 'enable_dynamic_creation'}
FUNCTION_BLOCK Node_F_VN_MaxElementElementwise_TcVnVector3_SINT EXTENDS VisionNode
VAR
    ipContainer : _ITcVnContainer;
    aMax : _TcVnVector3_SINT;
    hrPrev : _HRESULT(S_OK);
    hresult : _HRESULT(S_OK);
END_VAR

METHOD FB_init : BOOL
VAR_INPUT
	bInitRetains : BOOL; // if TRUE, the retain variables are initialized (warm start / cold start)
	bInCopyCode : BOOL;  // if TRUE, the instance afterwards gets moved into the copy code (online change)
END_VAR
AddInput('ipContainer', ipContainer);
AddInput('aMax', aMax);
AddInput('hrPrev', hrPrev);
AddOutput('ipContainer', ipContainer);
AddOutput('hresult',hresult);
END_METHOD

METHOD PUBLIC  Clone : I_Node
VAR
	pNode : POINTER TO Node_F_VN_MaxElementElementwise_TcVnVector3_SINT;
END_VAR
pNode := __NEW(Node_F_VN_MaxElementElementwise_TcVnVector3_SINT);
Clone := pNode^;
END_METHOD

METHOD PROTECTED OnExecute : HRESULT
hresult.Value := F_VN_MaxElementElementwise_TcVnVector3_SINT(
    ipContainer := ipContainer.Value,
    aMax := aMax.Value,
    hrPrev:= hrPrev.Value);
END_METHOD

METHOD PUBLIC PreExecutionCheck
VAR_INPUT
	Check : I_PreExecutionChecks;
END_VAR
Check.IsTrue(ipContainer.IsValid, 'ipContainer must be a valid container');
END_METHOD

END_FUNCTION_BLOCK

// Nodes/Container Statistics/Node_F_VN_MaxElementElementwise_TcVnVector3_UINT
{attribute 'linkalways'} 
{attribute 'no_explicit_call' := 'This FB is a CLASS and must be accessed using methods or properties'}
{attribute 'enable_dynamic_creation'}
FUNCTION_BLOCK Node_F_VN_MaxElementElementwise_TcVnVector3_UINT EXTENDS VisionNode
VAR
    ipContainer : _ITcVnContainer;
    aMax : _TcVnVector3_UINT;
    hrPrev : _HRESULT(S_OK);
    hresult : _HRESULT(S_OK);
END_VAR

METHOD FB_init : BOOL
VAR_INPUT
	bInitRetains : BOOL; // if TRUE, the retain variables are initialized (warm start / cold start)
	bInCopyCode : BOOL;  // if TRUE, the instance afterwards gets moved into the copy code (online change)
END_VAR
AddInput('ipContainer', ipContainer);
AddInput('aMax', aMax);
AddInput('hrPrev', hrPrev);
AddOutput('ipContainer', ipContainer);
AddOutput('hresult',hresult);
END_METHOD

METHOD PUBLIC  Clone : I_Node
VAR
	pNode : POINTER TO Node_F_VN_MaxElementElementwise_TcVnVector3_UINT;
END_VAR
pNode := __NEW(Node_F_VN_MaxElementElementwise_TcVnVector3_UINT);
Clone := pNode^;
END_METHOD

METHOD PROTECTED OnExecute : HRESULT
hresult.Value := F_VN_MaxElementElementwise_TcVnVector3_UINT(
    ipContainer := ipContainer.Value,
    aMax := aMax.Value,
    hrPrev:= hrPrev.Value);
END_METHOD

METHOD PUBLIC PreExecutionCheck
VAR_INPUT
	Check : I_PreExecutionChecks;
END_VAR
Check.IsTrue(ipContainer.IsValid, 'ipContainer must be a valid container');
END_METHOD

END_FUNCTION_BLOCK

// Nodes/Container Statistics/Node_F_VN_MaxElementElementwise_TcVnVector3_USINT
{attribute 'linkalways'} 
{attribute 'no_explicit_call' := 'This FB is a CLASS and must be accessed using methods or properties'}
{attribute 'enable_dynamic_creation'}
FUNCTION_BLOCK Node_F_VN_MaxElementElementwise_TcVnVector3_USINT EXTENDS VisionNode
VAR
    ipContainer : _ITcVnContainer;
    aMax : _TcVnVector3_USINT;
    hrPrev : _HRESULT(S_OK);
    hresult : _HRESULT(S_OK);
END_VAR

METHOD FB_init : BOOL
VAR_INPUT
	bInitRetains : BOOL; // if TRUE, the retain variables are initialized (warm start / cold start)
	bInCopyCode : BOOL;  // if TRUE, the instance afterwards gets moved into the copy code (online change)
END_VAR
AddInput('ipContainer', ipContainer);
AddInput('aMax', aMax);
AddInput('hrPrev', hrPrev);
AddOutput('ipContainer', ipContainer);
AddOutput('hresult',hresult);
END_METHOD

METHOD PUBLIC  Clone : I_Node
VAR
	pNode : POINTER TO Node_F_VN_MaxElementElementwise_TcVnVector3_USINT;
END_VAR
pNode := __NEW(Node_F_VN_MaxElementElementwise_TcVnVector3_USINT);
Clone := pNode^;
END_METHOD

METHOD PROTECTED OnExecute : HRESULT
hresult.Value := F_VN_MaxElementElementwise_TcVnVector3_USINT(
    ipContainer := ipContainer.Value,
    aMax := aMax.Value,
    hrPrev:= hrPrev.Value);
END_METHOD

METHOD PUBLIC PreExecutionCheck
VAR_INPUT
	Check : I_PreExecutionChecks;
END_VAR
Check.IsTrue(ipContainer.IsValid, 'ipContainer must be a valid container');
END_METHOD

END_FUNCTION_BLOCK

// Nodes/Container Statistics/Node_F_VN_MaxElementElementwise_TcVnVector4_DINT
{attribute 'linkalways'} 
{attribute 'no_explicit_call' := 'This FB is a CLASS and must be accessed using methods or properties'}
{attribute 'enable_dynamic_creation'}
FUNCTION_BLOCK Node_F_VN_MaxElementElementwise_TcVnVector4_DINT EXTENDS VisionNode
VAR
    ipContainer : _ITcVnContainer;
    aMax : _TcVnVector4_DINT;
    hrPrev : _HRESULT(S_OK);
    hresult : _HRESULT(S_OK);
END_VAR

METHOD FB_init : BOOL
VAR_INPUT
	bInitRetains : BOOL; // if TRUE, the retain variables are initialized (warm start / cold start)
	bInCopyCode : BOOL;  // if TRUE, the instance afterwards gets moved into the copy code (online change)
END_VAR
AddInput('ipContainer', ipContainer);
AddInput('aMax', aMax);
AddInput('hrPrev', hrPrev);
AddOutput('ipContainer', ipContainer);
AddOutput('hresult',hresult);
END_METHOD

METHOD PUBLIC  Clone : I_Node
VAR
	pNode : POINTER TO Node_F_VN_MaxElementElementwise_TcVnVector4_DINT;
END_VAR
pNode := __NEW(Node_F_VN_MaxElementElementwise_TcVnVector4_DINT);
Clone := pNode^;
END_METHOD

METHOD PROTECTED OnExecute : HRESULT
hresult.Value := F_VN_MaxElementElementwise_TcVnVector4_DINT(
    ipContainer := ipContainer.Value,
    aMax := aMax.Value,
    hrPrev:= hrPrev.Value);
END_METHOD

METHOD PUBLIC PreExecutionCheck
VAR_INPUT
	Check : I_PreExecutionChecks;
END_VAR
Check.IsTrue(ipContainer.IsValid, 'ipContainer must be a valid container');
END_METHOD

END_FUNCTION_BLOCK

// Nodes/Container Statistics/Node_F_VN_MaxElementElementwise_TcVnVector4_INT
{attribute 'linkalways'} 
{attribute 'no_explicit_call' := 'This FB is a CLASS and must be accessed using methods or properties'}
{attribute 'enable_dynamic_creation'}
FUNCTION_BLOCK Node_F_VN_MaxElementElementwise_TcVnVector4_INT EXTENDS VisionNode
VAR
    ipContainer : _ITcVnContainer;
    aMax : _TcVnVector4_INT;
    hrPrev : _HRESULT(S_OK);
    hresult : _HRESULT(S_OK);
END_VAR

METHOD FB_init : BOOL
VAR_INPUT
	bInitRetains : BOOL; // if TRUE, the retain variables are initialized (warm start / cold start)
	bInCopyCode : BOOL;  // if TRUE, the instance afterwards gets moved into the copy code (online change)
END_VAR
AddInput('ipContainer', ipContainer);
AddInput('aMax', aMax);
AddInput('hrPrev', hrPrev);
AddOutput('ipContainer', ipContainer);
AddOutput('hresult',hresult);
END_METHOD

METHOD PUBLIC  Clone : I_Node
VAR
	pNode : POINTER TO Node_F_VN_MaxElementElementwise_TcVnVector4_INT;
END_VAR
pNode := __NEW(Node_F_VN_MaxElementElementwise_TcVnVector4_INT);
Clone := pNode^;
END_METHOD

METHOD PROTECTED OnExecute : HRESULT
hresult.Value := F_VN_MaxElementElementwise_TcVnVector4_INT(
    ipContainer := ipContainer.Value,
    aMax := aMax.Value,
    hrPrev:= hrPrev.Value);
END_METHOD

METHOD PUBLIC PreExecutionCheck
VAR_INPUT
	Check : I_PreExecutionChecks;
END_VAR
Check.IsTrue(ipContainer.IsValid, 'ipContainer must be a valid container');
END_METHOD

END_FUNCTION_BLOCK

// Nodes/Container Statistics/Node_F_VN_MaxElementElementwise_TcVnVector4_LREAL
{attribute 'linkalways'} 
{attribute 'no_explicit_call' := 'This FB is a CLASS and must be accessed using methods or properties'}
{attribute 'enable_dynamic_creation'}
FUNCTION_BLOCK Node_F_VN_MaxElementElementwise_TcVnVector4_LREAL EXTENDS VisionNode
VAR
    ipContainer : _ITcVnContainer;
    aMax : _TcVnVector4_LREAL;
    hrPrev : _HRESULT(S_OK);
    hresult : _HRESULT(S_OK);
END_VAR

METHOD FB_init : BOOL
VAR_INPUT
	bInitRetains : BOOL; // if TRUE, the retain variables are initialized (warm start / cold start)
	bInCopyCode : BOOL;  // if TRUE, the instance afterwards gets moved into the copy code (online change)
END_VAR
AddInput('ipContainer', ipContainer);
AddInput('aMax', aMax);
AddInput('hrPrev', hrPrev);
AddOutput('ipContainer', ipContainer);
AddOutput('hresult',hresult);
END_METHOD

METHOD PUBLIC  Clone : I_Node
VAR
	pNode : POINTER TO Node_F_VN_MaxElementElementwise_TcVnVector4_LREAL;
END_VAR
pNode := __NEW(Node_F_VN_MaxElementElementwise_TcVnVector4_LREAL);
Clone := pNode^;
END_METHOD

METHOD PROTECTED OnExecute : HRESULT
hresult.Value := F_VN_MaxElementElementwise_TcVnVector4_LREAL(
    ipContainer := ipContainer.Value,
    aMax := aMax.Value,
    hrPrev:= hrPrev.Value);
END_METHOD

METHOD PUBLIC PreExecutionCheck
VAR_INPUT
	Check : I_PreExecutionChecks;
END_VAR
Check.IsTrue(ipContainer.IsValid, 'ipContainer must be a valid container');
END_METHOD

END_FUNCTION_BLOCK

// Nodes/Container Statistics/Node_F_VN_MaxElementElementwise_TcVnVector4_SINT
{attribute 'linkalways'} 
{attribute 'no_explicit_call' := 'This FB is a CLASS and must be accessed using methods or properties'}
{attribute 'enable_dynamic_creation'}
FUNCTION_BLOCK Node_F_VN_MaxElementElementwise_TcVnVector4_SINT EXTENDS VisionNode
VAR
    ipContainer : _ITcVnContainer;
    aMax : _TcVnVector4_SINT;
    hrPrev : _HRESULT(S_OK);
    hresult : _HRESULT(S_OK);
END_VAR

METHOD FB_init : BOOL
VAR_INPUT
	bInitRetains : BOOL; // if TRUE, the retain variables are initialized (warm start / cold start)
	bInCopyCode : BOOL;  // if TRUE, the instance afterwards gets moved into the copy code (online change)
END_VAR
AddInput('ipContainer', ipContainer);
AddInput('aMax', aMax);
AddInput('hrPrev', hrPrev);
AddOutput('ipContainer', ipContainer);
AddOutput('hresult',hresult);
END_METHOD

METHOD PUBLIC  Clone : I_Node
VAR
	pNode : POINTER TO Node_F_VN_MaxElementElementwise_TcVnVector4_SINT;
END_VAR
pNode := __NEW(Node_F_VN_MaxElementElementwise_TcVnVector4_SINT);
Clone := pNode^;
END_METHOD

METHOD PROTECTED OnExecute : HRESULT
hresult.Value := F_VN_MaxElementElementwise_TcVnVector4_SINT(
    ipContainer := ipContainer.Value,
    aMax := aMax.Value,
    hrPrev:= hrPrev.Value);
END_METHOD

METHOD PUBLIC PreExecutionCheck
VAR_INPUT
	Check : I_PreExecutionChecks;
END_VAR
Check.IsTrue(ipContainer.IsValid, 'ipContainer must be a valid container');
END_METHOD

END_FUNCTION_BLOCK

// Nodes/Container Statistics/Node_F_VN_MaxElementElementwise_TcVnVector4_UINT
{attribute 'linkalways'} 
{attribute 'no_explicit_call' := 'This FB is a CLASS and must be accessed using methods or properties'}
{attribute 'enable_dynamic_creation'}
FUNCTION_BLOCK Node_F_VN_MaxElementElementwise_TcVnVector4_UINT EXTENDS VisionNode
VAR
    ipContainer : _ITcVnContainer;
    aMax : _TcVnVector4_UINT;
    hrPrev : _HRESULT(S_OK);
    hresult : _HRESULT(S_OK);
END_VAR

METHOD FB_init : BOOL
VAR_INPUT
	bInitRetains : BOOL; // if TRUE, the retain variables are initialized (warm start / cold start)
	bInCopyCode : BOOL;  // if TRUE, the instance afterwards gets moved into the copy code (online change)
END_VAR
AddInput('ipContainer', ipContainer);
AddInput('aMax', aMax);
AddInput('hrPrev', hrPrev);
AddOutput('ipContainer', ipContainer);
AddOutput('hresult',hresult);
END_METHOD

METHOD PUBLIC  Clone : I_Node
VAR
	pNode : POINTER TO Node_F_VN_MaxElementElementwise_TcVnVector4_UINT;
END_VAR
pNode := __NEW(Node_F_VN_MaxElementElementwise_TcVnVector4_UINT);
Clone := pNode^;
END_METHOD

METHOD PROTECTED OnExecute : HRESULT
hresult.Value := F_VN_MaxElementElementwise_TcVnVector4_UINT(
    ipContainer := ipContainer.Value,
    aMax := aMax.Value,
    hrPrev:= hrPrev.Value);
END_METHOD

METHOD PUBLIC PreExecutionCheck
VAR_INPUT
	Check : I_PreExecutionChecks;
END_VAR
Check.IsTrue(ipContainer.IsValid, 'ipContainer must be a valid container');
END_METHOD

END_FUNCTION_BLOCK

// Nodes/Container Statistics/Node_F_VN_MaxElementElementwise_TcVnVector4_USINT
{attribute 'linkalways'} 
{attribute 'no_explicit_call' := 'This FB is a CLASS and must be accessed using methods or properties'}
{attribute 'enable_dynamic_creation'}
FUNCTION_BLOCK Node_F_VN_MaxElementElementwise_TcVnVector4_USINT EXTENDS VisionNode
VAR
    ipContainer : _ITcVnContainer;
    aMax : _TcVnVector4_USINT;
    hrPrev : _HRESULT(S_OK);
    hresult : _HRESULT(S_OK);
END_VAR

METHOD FB_init : BOOL
VAR_INPUT
	bInitRetains : BOOL; // if TRUE, the retain variables are initialized (warm start / cold start)
	bInCopyCode : BOOL;  // if TRUE, the instance afterwards gets moved into the copy code (online change)
END_VAR
AddInput('ipContainer', ipContainer);
AddInput('aMax', aMax);
AddInput('hrPrev', hrPrev);
AddOutput('ipContainer', ipContainer);
AddOutput('hresult',hresult);
END_METHOD

METHOD PUBLIC  Clone : I_Node
VAR
	pNode : POINTER TO Node_F_VN_MaxElementElementwise_TcVnVector4_USINT;
END_VAR
pNode := __NEW(Node_F_VN_MaxElementElementwise_TcVnVector4_USINT);
Clone := pNode^;
END_METHOD

METHOD PROTECTED OnExecute : HRESULT
hresult.Value := F_VN_MaxElementElementwise_TcVnVector4_USINT(
    ipContainer := ipContainer.Value,
    aMax := aMax.Value,
    hrPrev:= hrPrev.Value);
END_METHOD

METHOD PUBLIC PreExecutionCheck
VAR_INPUT
	Check : I_PreExecutionChecks;
END_VAR
Check.IsTrue(ipContainer.IsValid, 'ipContainer must be a valid container');
END_METHOD

END_FUNCTION_BLOCK

// Nodes/Container Statistics/Node_F_VN_MaxElementElementwise_UDINT
{attribute 'linkalways'} 
{attribute 'no_explicit_call' := 'This FB is a CLASS and must be accessed using methods or properties'}
{attribute 'enable_dynamic_creation'}
FUNCTION_BLOCK Node_F_VN_MaxElementElementwise_UDINT EXTENDS VisionNode
VAR
    ipContainer : _ITcVnContainer;
    nMax : _UDINT(0);
    hrPrev : _HRESULT(S_OK);
    hresult : _HRESULT(S_OK);
END_VAR

METHOD FB_init : BOOL
VAR_INPUT
	bInitRetains : BOOL; // if TRUE, the retain variables are initialized (warm start / cold start)
	bInCopyCode : BOOL;  // if TRUE, the instance afterwards gets moved into the copy code (online change)
END_VAR
AddInput('ipContainer', ipContainer);
AddInput('nMax', nMax);
AddInput('hrPrev', hrPrev);
AddOutput('ipContainer', ipContainer);
AddOutput('hresult',hresult);
END_METHOD

METHOD PUBLIC  Clone : I_Node
VAR
	pNode : POINTER TO Node_F_VN_MaxElementElementwise_UDINT;
END_VAR
pNode := __NEW(Node_F_VN_MaxElementElementwise_UDINT);
Clone := pNode^;
END_METHOD

METHOD PROTECTED OnExecute : HRESULT
hresult.Value := F_VN_MaxElementElementwise_UDINT(
    ipContainer := ipContainer.Value,
    nMax := nMax.Value,
    hrPrev:= hrPrev.Value);
END_METHOD

METHOD PUBLIC PreExecutionCheck
VAR_INPUT
	Check : I_PreExecutionChecks;
END_VAR
Check.IsTrue(ipContainer.IsValid, 'ipContainer must be a valid container');
Check.IsTrue(ipContainer.HasType('CTcVnContainer_Vector_UDINT'), 'ipContainer contains incorrect types');
END_METHOD

END_FUNCTION_BLOCK

// Nodes/Container Statistics/Node_F_VN_MaxElementElementwise_UINT
{attribute 'linkalways'} 
{attribute 'no_explicit_call' := 'This FB is a CLASS and must be accessed using methods or properties'}
{attribute 'enable_dynamic_creation'}
FUNCTION_BLOCK Node_F_VN_MaxElementElementwise_UINT EXTENDS VisionNode
VAR
    ipContainer : _ITcVnContainer;
    nMax : _UINT(0);
    hrPrev : _HRESULT(S_OK);
    hresult : _HRESULT(S_OK);
END_VAR

METHOD FB_init : BOOL
VAR_INPUT
	bInitRetains : BOOL; // if TRUE, the retain variables are initialized (warm start / cold start)
	bInCopyCode : BOOL;  // if TRUE, the instance afterwards gets moved into the copy code (online change)
END_VAR
AddInput('ipContainer', ipContainer);
AddInput('nMax', nMax);
AddInput('hrPrev', hrPrev);
AddOutput('ipContainer', ipContainer);
AddOutput('hresult',hresult);
END_METHOD

METHOD PUBLIC  Clone : I_Node
VAR
	pNode : POINTER TO Node_F_VN_MaxElementElementwise_UINT;
END_VAR
pNode := __NEW(Node_F_VN_MaxElementElementwise_UINT);
Clone := pNode^;
END_METHOD

METHOD PROTECTED OnExecute : HRESULT
hresult.Value := F_VN_MaxElementElementwise_UINT(
    ipContainer := ipContainer.Value,
    nMax := nMax.Value,
    hrPrev:= hrPrev.Value);
END_METHOD

METHOD PUBLIC PreExecutionCheck
VAR_INPUT
	Check : I_PreExecutionChecks;
END_VAR
Check.IsTrue(ipContainer.IsValid, 'ipContainer must be a valid container');
Check.IsTrue(ipContainer.HasType('CTcVnContainer_Vector_UDINT'), 'ipContainer contains incorrect types');
END_METHOD

END_FUNCTION_BLOCK

// Nodes/Container Statistics/Node_F_VN_MaxElementElementwise_ULINT
{attribute 'linkalways'} 
{attribute 'no_explicit_call' := 'This FB is a CLASS and must be accessed using methods or properties'}
{attribute 'enable_dynamic_creation'}
FUNCTION_BLOCK Node_F_VN_MaxElementElementwise_ULINT EXTENDS VisionNode
VAR
    ipContainer : _ITcVnContainer;
    nMax : _ULINT(0);
    hrPrev : _HRESULT(S_OK);
    hresult : _HRESULT(S_OK);
END_VAR

METHOD FB_init : BOOL
VAR_INPUT
	bInitRetains : BOOL; // if TRUE, the retain variables are initialized (warm start / cold start)
	bInCopyCode : BOOL;  // if TRUE, the instance afterwards gets moved into the copy code (online change)
END_VAR
AddInput('ipContainer', ipContainer);
AddInput('nMax', nMax);
AddInput('hrPrev', hrPrev);
AddOutput('ipContainer', ipContainer);
AddOutput('hresult',hresult);
END_METHOD

METHOD PUBLIC  Clone : I_Node
VAR
	pNode : POINTER TO Node_F_VN_MaxElementElementwise_ULINT;
END_VAR
pNode := __NEW(Node_F_VN_MaxElementElementwise_ULINT);
Clone := pNode^;
END_METHOD

METHOD PROTECTED OnExecute : HRESULT
hresult.Value := F_VN_MaxElementElementwise_ULINT(
    ipContainer := ipContainer.Value,
    nMax := nMax.Value,
    hrPrev:= hrPrev.Value);
END_METHOD

METHOD PUBLIC PreExecutionCheck
VAR_INPUT
	Check : I_PreExecutionChecks;
END_VAR
Check.IsTrue(ipContainer.IsValid, 'ipContainer must be a valid container');
Check.IsTrue(ipContainer.HasType('CTcVnContainer_Vector_ULINT'), 'ipContainer contains incorrect types');
END_METHOD

END_FUNCTION_BLOCK

// Nodes/Container Statistics/Node_F_VN_MaxElementElementwise_USINT
{attribute 'linkalways'} 
{attribute 'no_explicit_call' := 'This FB is a CLASS and must be accessed using methods or properties'}
{attribute 'enable_dynamic_creation'}
FUNCTION_BLOCK Node_F_VN_MaxElementElementwise_USINT EXTENDS VisionNode
VAR
    ipContainer : _ITcVnContainer;
    nMax : _USINT(0);
    hrPrev : _HRESULT(S_OK);
    hresult : _HRESULT(S_OK);
END_VAR

METHOD FB_init : BOOL
VAR_INPUT
	bInitRetains : BOOL; // if TRUE, the retain variables are initialized (warm start / cold start)
	bInCopyCode : BOOL;  // if TRUE, the instance afterwards gets moved into the copy code (online change)
END_VAR
AddInput('ipContainer', ipContainer);
AddInput('nMax', nMax);
AddInput('hrPrev', hrPrev);
AddOutput('ipContainer', ipContainer);
AddOutput('hresult',hresult);
END_METHOD

METHOD PUBLIC  Clone : I_Node
VAR
	pNode : POINTER TO Node_F_VN_MaxElementElementwise_USINT;
END_VAR
pNode := __NEW(Node_F_VN_MaxElementElementwise_USINT);
Clone := pNode^;
END_METHOD

METHOD PROTECTED OnExecute : HRESULT
hresult.Value := F_VN_MaxElementElementwise_USINT(
    ipContainer := ipContainer.Value,
    nMax := nMax.Value,
    hrPrev:= hrPrev.Value);
END_METHOD

METHOD PUBLIC PreExecutionCheck
VAR_INPUT
	Check : I_PreExecutionChecks;
END_VAR
Check.IsTrue(ipContainer.IsValid, 'ipContainer must be a valid container');
Check.IsTrue(ipContainer.HasType('CTcVnContainer_Vector_USINT'), 'ipContainer contains incorrect types');
END_METHOD

END_FUNCTION_BLOCK

// Nodes/Container Statistics/Node_F_VN_MedianElementElementwise_DINT
{attribute 'linkalways'} 
{attribute 'no_explicit_call' := 'This FB is a CLASS and must be accessed using methods or properties'}
{attribute 'enable_dynamic_creation'}
FUNCTION_BLOCK Node_F_VN_MedianElementElementwise_DINT EXTENDS VisionNode
VAR
    ipContainer : _ITcVnContainer;
    nMedian : _DINT(0);
    hrPrev : _HRESULT(S_OK);
    hresult : _HRESULT(S_OK);
END_VAR

METHOD FB_init : BOOL
VAR_INPUT
	bInitRetains : BOOL; // if TRUE, the retain variables are initialized (warm start / cold start)
	bInCopyCode : BOOL;  // if TRUE, the instance afterwards gets moved into the copy code (online change)
END_VAR
AddInput('ipContainer', ipContainer);
AddInput('nMedian', nMedian);
AddInput('hrPrev', hrPrev);
AddOutput('ipContainer', ipContainer);
AddOutput('hresult',hresult);
END_METHOD

METHOD PUBLIC  Clone : I_Node
VAR
	pNode : POINTER TO Node_F_VN_MedianElementElementwise_DINT;
END_VAR
pNode := __NEW(Node_F_VN_MedianElementElementwise_DINT);
Clone := pNode^;
END_METHOD

METHOD PROTECTED OnExecute : HRESULT
hresult.Value := F_VN_MedianElementElementwise_DINT(
    ipContainer := ipContainer.Value,
    nMedian := nMedian.Value,
    hrPrev:= hrPrev.Value);
END_METHOD

METHOD PUBLIC PreExecutionCheck
VAR_INPUT
	Check : I_PreExecutionChecks;
END_VAR
Check.IsTrue(ipContainer.IsValid, 'ipContainer must be a valid container');
Check.IsTrue(ipContainer.HasType('CTcVnContainer_Vector_DINT'), 'ipContainer contains incorrect types');
END_METHOD

END_FUNCTION_BLOCK

// Nodes/Container Statistics/Node_F_VN_MedianElementElementwise_INT
{attribute 'linkalways'} 
{attribute 'no_explicit_call' := 'This FB is a CLASS and must be accessed using methods or properties'}
{attribute 'enable_dynamic_creation'}
FUNCTION_BLOCK Node_F_VN_MedianElementElementwise_INT EXTENDS VisionNode
VAR
    ipContainer : _ITcVnContainer;
    nMedian : _INT(0);
    hrPrev : _HRESULT(S_OK);
    hresult : _HRESULT(S_OK);
END_VAR

METHOD FB_init : BOOL
VAR_INPUT
	bInitRetains : BOOL; // if TRUE, the retain variables are initialized (warm start / cold start)
	bInCopyCode : BOOL;  // if TRUE, the instance afterwards gets moved into the copy code (online change)
END_VAR
AddInput('ipContainer', ipContainer);
AddInput('nMedian', nMedian);
AddInput('hrPrev', hrPrev);
AddOutput('ipContainer', ipContainer);
AddOutput('hresult',hresult);
END_METHOD

METHOD PUBLIC  Clone : I_Node
VAR
	pNode : POINTER TO Node_F_VN_MedianElementElementwise_INT;
END_VAR
pNode := __NEW(Node_F_VN_MedianElementElementwise_INT);
Clone := pNode^;
END_METHOD

METHOD PROTECTED OnExecute : HRESULT
hresult.Value := F_VN_MedianElementElementwise_INT(
    ipContainer := ipContainer.Value,
    nMedian := nMedian.Value,
    hrPrev:= hrPrev.Value);
END_METHOD

METHOD PUBLIC PreExecutionCheck
VAR_INPUT
	Check : I_PreExecutionChecks;
END_VAR
Check.IsTrue(ipContainer.IsValid, 'ipContainer must be a valid container');
Check.IsTrue(ipContainer.HasType('CTcVnContainer_Vector_INT'), 'ipContainer contains incorrect types');
END_METHOD

END_FUNCTION_BLOCK

// Nodes/Container Statistics/Node_F_VN_MedianElementElementwise_LREAL
{attribute 'linkalways'} 
{attribute 'no_explicit_call' := 'This FB is a CLASS and must be accessed using methods or properties'}
{attribute 'enable_dynamic_creation'}
FUNCTION_BLOCK Node_F_VN_MedianElementElementwise_LREAL EXTENDS VisionNode
VAR
    ipContainer : _ITcVnContainer;
    fMedian : _LREAL(0.0);
    hrPrev : _HRESULT(S_OK);
    hresult : _HRESULT(S_OK);
END_VAR

METHOD FB_init : BOOL
VAR_INPUT
	bInitRetains : BOOL; // if TRUE, the retain variables are initialized (warm start / cold start)
	bInCopyCode : BOOL;  // if TRUE, the instance afterwards gets moved into the copy code (online change)
END_VAR
AddInput('ipContainer', ipContainer);
AddInput('fMedian', fMedian);
AddInput('hrPrev', hrPrev);
AddOutput('ipContainer', ipContainer);
AddOutput('hresult',hresult);
END_METHOD

METHOD PUBLIC  Clone : I_Node
VAR
	pNode : POINTER TO Node_F_VN_MedianElementElementwise_LREAL;
END_VAR
pNode := __NEW(Node_F_VN_MedianElementElementwise_LREAL);
Clone := pNode^;
END_METHOD

METHOD PROTECTED OnExecute : HRESULT
hresult.Value := F_VN_MedianElementElementwise_LREAL(
    ipContainer := ipContainer.Value,
    fMedian := fMedian.Value,
    hrPrev:= hrPrev.Value);
END_METHOD

METHOD PUBLIC PreExecutionCheck
VAR_INPUT
	Check : I_PreExecutionChecks;
END_VAR
Check.IsTrue(ipContainer.IsValid, 'ipContainer must be a valid container');
Check.IsTrue(ipContainer.HasType('CTcVnContainer_Vector_LREAL'), 'ipContainer contains incorrect types');
END_METHOD

END_FUNCTION_BLOCK

// Nodes/Container Statistics/Node_F_VN_MedianElementElementwise_REAL
{attribute 'linkalways'} 
{attribute 'no_explicit_call' := 'This FB is a CLASS and must be accessed using methods or properties'}
{attribute 'enable_dynamic_creation'}
FUNCTION_BLOCK Node_F_VN_MedianElementElementwise_REAL EXTENDS VisionNode
VAR
    ipContainer : _ITcVnContainer;
    fMedian : _REAL(0.0);
    hrPrev : _HRESULT(S_OK);
    hresult : _HRESULT(S_OK);
END_VAR

METHOD FB_init : BOOL
VAR_INPUT
	bInitRetains : BOOL; // if TRUE, the retain variables are initialized (warm start / cold start)
	bInCopyCode : BOOL;  // if TRUE, the instance afterwards gets moved into the copy code (online change)
END_VAR
AddInput('ipContainer', ipContainer);
AddInput('fMedian', fMedian);
AddInput('hrPrev', hrPrev);
AddOutput('ipContainer', ipContainer);
AddOutput('hresult',hresult);
END_METHOD

METHOD PUBLIC  Clone : I_Node
VAR
	pNode : POINTER TO Node_F_VN_MedianElementElementwise_REAL;
END_VAR
pNode := __NEW(Node_F_VN_MedianElementElementwise_REAL);
Clone := pNode^;
END_METHOD

METHOD PROTECTED OnExecute : HRESULT
hresult.Value := F_VN_MedianElementElementwise_REAL(
    ipContainer := ipContainer.Value,
    fMedian := fMedian.Value,
    hrPrev:= hrPrev.Value);
END_METHOD

METHOD PUBLIC PreExecutionCheck
VAR_INPUT
	Check : I_PreExecutionChecks;
END_VAR
Check.IsTrue(ipContainer.IsValid, 'ipContainer must be a valid container');
Check.IsTrue(ipContainer.HasType('CTcVnContainer_Vector_REAL'), 'ipContainer contains incorrect types');
END_METHOD

END_FUNCTION_BLOCK

// Nodes/Container Statistics/Node_F_VN_MedianElementElementwise_SINT
{attribute 'linkalways'} 
{attribute 'no_explicit_call' := 'This FB is a CLASS and must be accessed using methods or properties'}
{attribute 'enable_dynamic_creation'}
FUNCTION_BLOCK Node_F_VN_MedianElementElementwise_SINT EXTENDS VisionNode
VAR
    ipContainer : _ITcVnContainer;
    nMedian : _SINT(0);
    hrPrev : _HRESULT(S_OK);
    hresult : _HRESULT(S_OK);
END_VAR

METHOD FB_init : BOOL
VAR_INPUT
	bInitRetains : BOOL; // if TRUE, the retain variables are initialized (warm start / cold start)
	bInCopyCode : BOOL;  // if TRUE, the instance afterwards gets moved into the copy code (online change)
END_VAR
AddInput('ipContainer', ipContainer);
AddInput('nMedian', nMedian);
AddInput('hrPrev', hrPrev);
AddOutput('ipContainer', ipContainer);
AddOutput('hresult',hresult);
END_METHOD

METHOD PUBLIC  Clone : I_Node
VAR
	pNode : POINTER TO Node_F_VN_MedianElementElementwise_SINT;
END_VAR
pNode := __NEW(Node_F_VN_MedianElementElementwise_SINT);
Clone := pNode^;
END_METHOD

METHOD PROTECTED OnExecute : HRESULT
hresult.Value := F_VN_MedianElementElementwise_SINT(
    ipContainer := ipContainer.Value,
    nMedian := nMedian.Value,
    hrPrev:= hrPrev.Value);
END_METHOD

METHOD PUBLIC PreExecutionCheck
VAR_INPUT
	Check : I_PreExecutionChecks;
END_VAR
Check.IsTrue(ipContainer.IsValid, 'ipContainer must be a valid container');
Check.IsTrue(ipContainer.HasType('CTcVnContainer_Vector_SINT'), 'ipContainer contains incorrect types');
END_METHOD

END_FUNCTION_BLOCK

// Nodes/Container Statistics/Node_F_VN_MedianElementElementwise_TcVnPoint2_DINT
{attribute 'linkalways'} 
{attribute 'no_explicit_call' := 'This FB is a CLASS and must be accessed using methods or properties'}
{attribute 'enable_dynamic_creation'}
FUNCTION_BLOCK Node_F_VN_MedianElementElementwise_TcVnPoint2_DINT EXTENDS VisionNode
VAR
    ipContainer : _ITcVnContainer;
    aMedian : _TcVnPoint2_DINT;
    hrPrev : _HRESULT(S_OK);
    hresult : _HRESULT(S_OK);
END_VAR

METHOD FB_init : BOOL
VAR_INPUT
	bInitRetains : BOOL; // if TRUE, the retain variables are initialized (warm start / cold start)
	bInCopyCode : BOOL;  // if TRUE, the instance afterwards gets moved into the copy code (online change)
END_VAR
AddInput('ipContainer', ipContainer);
AddInput('aMedian', aMedian);
AddInput('hrPrev', hrPrev);
AddOutput('ipContainer', ipContainer);
AddOutput('hresult',hresult);
END_METHOD

METHOD PUBLIC  Clone : I_Node
VAR
	pNode : POINTER TO Node_F_VN_MedianElementElementwise_TcVnPoint2_DINT;
END_VAR
pNode := __NEW(Node_F_VN_MedianElementElementwise_TcVnPoint2_DINT);
Clone := pNode^;
END_METHOD

METHOD PROTECTED OnExecute : HRESULT
hresult.Value := F_VN_MedianElementElementwise_TcVnPoint2_DINT(
    ipContainer := ipContainer.Value,
    aMedian := aMedian.Value,
    hrPrev:= hrPrev.Value);
END_METHOD

METHOD PUBLIC PreExecutionCheck
VAR_INPUT
	Check : I_PreExecutionChecks;
END_VAR
Check.IsTrue(ipContainer.IsValid, 'ipContainer must be a valid container');
END_METHOD

END_FUNCTION_BLOCK

// Nodes/Container Statistics/Node_F_VN_MedianElementElementwise_TcVnPoint2_LREAL
{attribute 'linkalways'} 
{attribute 'no_explicit_call' := 'This FB is a CLASS and must be accessed using methods or properties'}
{attribute 'enable_dynamic_creation'}
FUNCTION_BLOCK Node_F_VN_MedianElementElementwise_TcVnPoint2_LREAL EXTENDS VisionNode
VAR
    ipContainer : _ITcVnContainer;
    aMedian : _TcVnPoint2_LREAL;
    hrPrev : _HRESULT(S_OK);
    hresult : _HRESULT(S_OK);
END_VAR

METHOD FB_init : BOOL
VAR_INPUT
	bInitRetains : BOOL; // if TRUE, the retain variables are initialized (warm start / cold start)
	bInCopyCode : BOOL;  // if TRUE, the instance afterwards gets moved into the copy code (online change)
END_VAR
AddInput('ipContainer', ipContainer);
AddInput('aMedian', aMedian);
AddInput('hrPrev', hrPrev);
AddOutput('ipContainer', ipContainer);
AddOutput('hresult',hresult);
END_METHOD

METHOD PUBLIC  Clone : I_Node
VAR
	pNode : POINTER TO Node_F_VN_MedianElementElementwise_TcVnPoint2_LREAL;
END_VAR
pNode := __NEW(Node_F_VN_MedianElementElementwise_TcVnPoint2_LREAL);
Clone := pNode^;
END_METHOD

METHOD PROTECTED OnExecute : HRESULT
hresult.Value := F_VN_MedianElementElementwise_TcVnPoint2_LREAL(
    ipContainer := ipContainer.Value,
    aMedian := aMedian.Value,
    hrPrev:= hrPrev.Value);
END_METHOD

METHOD PUBLIC PreExecutionCheck
VAR_INPUT
	Check : I_PreExecutionChecks;
END_VAR
Check.IsTrue(ipContainer.IsValid, 'ipContainer must be a valid container');
END_METHOD

END_FUNCTION_BLOCK

// Nodes/Container Statistics/Node_F_VN_MedianElementElementwise_TcVnPoint2_REAL
{attribute 'linkalways'} 
{attribute 'no_explicit_call' := 'This FB is a CLASS and must be accessed using methods or properties'}
{attribute 'enable_dynamic_creation'}
FUNCTION_BLOCK Node_F_VN_MedianElementElementwise_TcVnPoint2_REAL EXTENDS VisionNode
VAR
    ipContainer : _ITcVnContainer;
    aMedian : _TcVnPoint2_REAL;
    hrPrev : _HRESULT(S_OK);
    hresult : _HRESULT(S_OK);
END_VAR

METHOD FB_init : BOOL
VAR_INPUT
	bInitRetains : BOOL; // if TRUE, the retain variables are initialized (warm start / cold start)
	bInCopyCode : BOOL;  // if TRUE, the instance afterwards gets moved into the copy code (online change)
END_VAR
AddInput('ipContainer', ipContainer);
AddInput('aMedian', aMedian);
AddInput('hrPrev', hrPrev);
AddOutput('ipContainer', ipContainer);
AddOutput('hresult',hresult);
END_METHOD

METHOD PUBLIC  Clone : I_Node
VAR
	pNode : POINTER TO Node_F_VN_MedianElementElementwise_TcVnPoint2_REAL;
END_VAR
pNode := __NEW(Node_F_VN_MedianElementElementwise_TcVnPoint2_REAL);
Clone := pNode^;
END_METHOD

METHOD PROTECTED OnExecute : HRESULT
hresult.Value := F_VN_MedianElementElementwise_TcVnPoint2_REAL(
    ipContainer := ipContainer.Value,
    aMedian := aMedian.Value,
    hrPrev:= hrPrev.Value);
END_METHOD

METHOD PUBLIC PreExecutionCheck
VAR_INPUT
	Check : I_PreExecutionChecks;
END_VAR
Check.IsTrue(ipContainer.IsValid, 'ipContainer must be a valid container');
END_METHOD

END_FUNCTION_BLOCK

// Nodes/Container Statistics/Node_F_VN_MedianElementElementwise_TcVnPoint3_LREAL
{attribute 'linkalways'} 
{attribute 'no_explicit_call' := 'This FB is a CLASS and must be accessed using methods or properties'}
{attribute 'enable_dynamic_creation'}
FUNCTION_BLOCK Node_F_VN_MedianElementElementwise_TcVnPoint3_LREAL EXTENDS VisionNode
VAR
    ipContainer : _ITcVnContainer;
    aMedian : _TcVnPoint3_LREAL;
    hrPrev : _HRESULT(S_OK);
    hresult : _HRESULT(S_OK);
END_VAR

METHOD FB_init : BOOL
VAR_INPUT
	bInitRetains : BOOL; // if TRUE, the retain variables are initialized (warm start / cold start)
	bInCopyCode : BOOL;  // if TRUE, the instance afterwards gets moved into the copy code (online change)
END_VAR
AddInput('ipContainer', ipContainer);
AddInput('aMedian', aMedian);
AddInput('hrPrev', hrPrev);
AddOutput('ipContainer', ipContainer);
AddOutput('hresult',hresult);
END_METHOD

METHOD PUBLIC  Clone : I_Node
VAR
	pNode : POINTER TO Node_F_VN_MedianElementElementwise_TcVnPoint3_LREAL;
END_VAR
pNode := __NEW(Node_F_VN_MedianElementElementwise_TcVnPoint3_LREAL);
Clone := pNode^;
END_METHOD

METHOD PROTECTED OnExecute : HRESULT
hresult.Value := F_VN_MedianElementElementwise_TcVnPoint3_LREAL(
    ipContainer := ipContainer.Value,
    aMedian := aMedian.Value,
    hrPrev:= hrPrev.Value);
END_METHOD

METHOD PUBLIC PreExecutionCheck
VAR_INPUT
	Check : I_PreExecutionChecks;
END_VAR
Check.IsTrue(ipContainer.IsValid, 'ipContainer must be a valid container');
END_METHOD

END_FUNCTION_BLOCK

// Nodes/Container Statistics/Node_F_VN_MedianElementElementwise_TcVnPoint3_REAL
{attribute 'linkalways'} 
{attribute 'no_explicit_call' := 'This FB is a CLASS and must be accessed using methods or properties'}
{attribute 'enable_dynamic_creation'}
FUNCTION_BLOCK Node_F_VN_MedianElementElementwise_TcVnPoint3_REAL EXTENDS VisionNode
VAR
    ipContainer : _ITcVnContainer;
    aMedian : _TcVnPoint3_REAL;
    hrPrev : _HRESULT(S_OK);
    hresult : _HRESULT(S_OK);
END_VAR

METHOD FB_init : BOOL
VAR_INPUT
	bInitRetains : BOOL; // if TRUE, the retain variables are initialized (warm start / cold start)
	bInCopyCode : BOOL;  // if TRUE, the instance afterwards gets moved into the copy code (online change)
END_VAR
AddInput('ipContainer', ipContainer);
AddInput('aMedian', aMedian);
AddInput('hrPrev', hrPrev);
AddOutput('ipContainer', ipContainer);
AddOutput('hresult',hresult);
END_METHOD

METHOD PUBLIC  Clone : I_Node
VAR
	pNode : POINTER TO Node_F_VN_MedianElementElementwise_TcVnPoint3_REAL;
END_VAR
pNode := __NEW(Node_F_VN_MedianElementElementwise_TcVnPoint3_REAL);
Clone := pNode^;
END_METHOD

METHOD PROTECTED OnExecute : HRESULT
hresult.Value := F_VN_MedianElementElementwise_TcVnPoint3_REAL(
    ipContainer := ipContainer.Value,
    aMedian := aMedian.Value,
    hrPrev:= hrPrev.Value);
END_METHOD

METHOD PUBLIC PreExecutionCheck
VAR_INPUT
	Check : I_PreExecutionChecks;
END_VAR
Check.IsTrue(ipContainer.IsValid, 'ipContainer must be a valid container');
END_METHOD

END_FUNCTION_BLOCK

// Nodes/Container Statistics/Node_F_VN_MedianElementElementwise_TcVnVector2_DINT
{attribute 'linkalways'} 
{attribute 'no_explicit_call' := 'This FB is a CLASS and must be accessed using methods or properties'}
{attribute 'enable_dynamic_creation'}
FUNCTION_BLOCK Node_F_VN_MedianElementElementwise_TcVnVector2_DINT EXTENDS VisionNode
VAR
    ipContainer : _ITcVnContainer;
    aMedian : _TcVnVector2_DINT;
    hrPrev : _HRESULT(S_OK);
    hresult : _HRESULT(S_OK);
END_VAR

METHOD FB_init : BOOL
VAR_INPUT
	bInitRetains : BOOL; // if TRUE, the retain variables are initialized (warm start / cold start)
	bInCopyCode : BOOL;  // if TRUE, the instance afterwards gets moved into the copy code (online change)
END_VAR
AddInput('ipContainer', ipContainer);
AddInput('aMedian', aMedian);
AddInput('hrPrev', hrPrev);
AddOutput('ipContainer', ipContainer);
AddOutput('hresult',hresult);
END_METHOD

METHOD PUBLIC  Clone : I_Node
VAR
	pNode : POINTER TO Node_F_VN_MedianElementElementwise_TcVnVector2_DINT;
END_VAR
pNode := __NEW(Node_F_VN_MedianElementElementwise_TcVnVector2_DINT);
Clone := pNode^;
END_METHOD

METHOD PROTECTED OnExecute : HRESULT
hresult.Value := F_VN_MedianElementElementwise_TcVnVector2_DINT(
    ipContainer := ipContainer.Value,
    aMedian := aMedian.Value,
    hrPrev:= hrPrev.Value);
END_METHOD

METHOD PUBLIC PreExecutionCheck
VAR_INPUT
	Check : I_PreExecutionChecks;
END_VAR
Check.IsTrue(ipContainer.IsValid, 'ipContainer must be a valid container');
END_METHOD

END_FUNCTION_BLOCK

// Nodes/Container Statistics/Node_F_VN_MedianElementElementwise_TcVnVector2_INT
{attribute 'linkalways'} 
{attribute 'no_explicit_call' := 'This FB is a CLASS and must be accessed using methods or properties'}
{attribute 'enable_dynamic_creation'}
FUNCTION_BLOCK Node_F_VN_MedianElementElementwise_TcVnVector2_INT EXTENDS VisionNode
VAR
    ipContainer : _ITcVnContainer;
    aMedian : _TcVnVector2_INT;
    hrPrev : _HRESULT(S_OK);
    hresult : _HRESULT(S_OK);
END_VAR

METHOD FB_init : BOOL
VAR_INPUT
	bInitRetains : BOOL; // if TRUE, the retain variables are initialized (warm start / cold start)
	bInCopyCode : BOOL;  // if TRUE, the instance afterwards gets moved into the copy code (online change)
END_VAR
AddInput('ipContainer', ipContainer);
AddInput('aMedian', aMedian);
AddInput('hrPrev', hrPrev);
AddOutput('ipContainer', ipContainer);
AddOutput('hresult',hresult);
END_METHOD

METHOD PUBLIC  Clone : I_Node
VAR
	pNode : POINTER TO Node_F_VN_MedianElementElementwise_TcVnVector2_INT;
END_VAR
pNode := __NEW(Node_F_VN_MedianElementElementwise_TcVnVector2_INT);
Clone := pNode^;
END_METHOD

METHOD PROTECTED OnExecute : HRESULT
hresult.Value := F_VN_MedianElementElementwise_TcVnVector2_INT(
    ipContainer := ipContainer.Value,
    aMedian := aMedian.Value,
    hrPrev:= hrPrev.Value);
END_METHOD

METHOD PUBLIC PreExecutionCheck
VAR_INPUT
	Check : I_PreExecutionChecks;
END_VAR
Check.IsTrue(ipContainer.IsValid, 'ipContainer must be a valid container');
END_METHOD

END_FUNCTION_BLOCK

// Nodes/Container Statistics/Node_F_VN_MedianElementElementwise_TcVnVector2_REAL
{attribute 'linkalways'} 
{attribute 'no_explicit_call' := 'This FB is a CLASS and must be accessed using methods or properties'}
{attribute 'enable_dynamic_creation'}
FUNCTION_BLOCK Node_F_VN_MedianElementElementwise_TcVnVector2_REAL EXTENDS VisionNode
VAR
    ipContainer : _ITcVnContainer;
    aMedian : _TcVnVector2_REAL;
    hrPrev : _HRESULT(S_OK);
    hresult : _HRESULT(S_OK);
END_VAR

METHOD FB_init : BOOL
VAR_INPUT
	bInitRetains : BOOL; // if TRUE, the retain variables are initialized (warm start / cold start)
	bInCopyCode : BOOL;  // if TRUE, the instance afterwards gets moved into the copy code (online change)
END_VAR
AddInput('ipContainer', ipContainer);
AddInput('aMedian', aMedian);
AddInput('hrPrev', hrPrev);
AddOutput('ipContainer', ipContainer);
AddOutput('hresult',hresult);
END_METHOD

METHOD PUBLIC  Clone : I_Node
VAR
	pNode : POINTER TO Node_F_VN_MedianElementElementwise_TcVnVector2_REAL;
END_VAR
pNode := __NEW(Node_F_VN_MedianElementElementwise_TcVnVector2_REAL);
Clone := pNode^;
END_METHOD

METHOD PROTECTED OnExecute : HRESULT
hresult.Value := F_VN_MedianElementElementwise_TcVnVector2_REAL(
    ipContainer := ipContainer.Value,
    aMedian := aMedian.Value,
    hrPrev:= hrPrev.Value);
END_METHOD

METHOD PUBLIC PreExecutionCheck
VAR_INPUT
	Check : I_PreExecutionChecks;
END_VAR
Check.IsTrue(ipContainer.IsValid, 'ipContainer must be a valid container');
END_METHOD

END_FUNCTION_BLOCK

// Nodes/Container Statistics/Node_F_VN_MedianElementElementwise_TcVnVector2_SINT
{attribute 'linkalways'} 
{attribute 'no_explicit_call' := 'This FB is a CLASS and must be accessed using methods or properties'}
{attribute 'enable_dynamic_creation'}
FUNCTION_BLOCK Node_F_VN_MedianElementElementwise_TcVnVector2_SINT EXTENDS VisionNode
VAR
    ipContainer : _ITcVnContainer;
    aMedian : _TcVnVector2_SINT;
    hrPrev : _HRESULT(S_OK);
    hresult : _HRESULT(S_OK);
END_VAR

METHOD FB_init : BOOL
VAR_INPUT
	bInitRetains : BOOL; // if TRUE, the retain variables are initialized (warm start / cold start)
	bInCopyCode : BOOL;  // if TRUE, the instance afterwards gets moved into the copy code (online change)
END_VAR
AddInput('ipContainer', ipContainer);
AddInput('aMedian', aMedian);
AddInput('hrPrev', hrPrev);
AddOutput('ipContainer', ipContainer);
AddOutput('hresult',hresult);
END_METHOD

METHOD PUBLIC  Clone : I_Node
VAR
	pNode : POINTER TO Node_F_VN_MedianElementElementwise_TcVnVector2_SINT;
END_VAR
pNode := __NEW(Node_F_VN_MedianElementElementwise_TcVnVector2_SINT);
Clone := pNode^;
END_METHOD

METHOD PROTECTED OnExecute : HRESULT
hresult.Value := F_VN_MedianElementElementwise_TcVnVector2_SINT(
    ipContainer := ipContainer.Value,
    aMedian := aMedian.Value,
    hrPrev:= hrPrev.Value);
END_METHOD

METHOD PUBLIC PreExecutionCheck
VAR_INPUT
	Check : I_PreExecutionChecks;
END_VAR
Check.IsTrue(ipContainer.IsValid, 'ipContainer must be a valid container');
END_METHOD

END_FUNCTION_BLOCK

// Nodes/Container Statistics/Node_F_VN_MedianElementElementwise_TcVnVector2_UINT
{attribute 'linkalways'} 
{attribute 'no_explicit_call' := 'This FB is a CLASS and must be accessed using methods or properties'}
{attribute 'enable_dynamic_creation'}
FUNCTION_BLOCK Node_F_VN_MedianElementElementwise_TcVnVector2_UINT EXTENDS VisionNode
VAR
    ipContainer : _ITcVnContainer;
    aMedian : _TcVnVector2_UINT;
    hrPrev : _HRESULT(S_OK);
    hresult : _HRESULT(S_OK);
END_VAR

METHOD FB_init : BOOL
VAR_INPUT
	bInitRetains : BOOL; // if TRUE, the retain variables are initialized (warm start / cold start)
	bInCopyCode : BOOL;  // if TRUE, the instance afterwards gets moved into the copy code (online change)
END_VAR
AddInput('ipContainer', ipContainer);
AddInput('aMedian', aMedian);
AddInput('hrPrev', hrPrev);
AddOutput('ipContainer', ipContainer);
AddOutput('hresult',hresult);
END_METHOD

METHOD PUBLIC  Clone : I_Node
VAR
	pNode : POINTER TO Node_F_VN_MedianElementElementwise_TcVnVector2_UINT;
END_VAR
pNode := __NEW(Node_F_VN_MedianElementElementwise_TcVnVector2_UINT);
Clone := pNode^;
END_METHOD

METHOD PROTECTED OnExecute : HRESULT
hresult.Value := F_VN_MedianElementElementwise_TcVnVector2_UINT(
    ipContainer := ipContainer.Value,
    aMedian := aMedian.Value,
    hrPrev:= hrPrev.Value);
END_METHOD

METHOD PUBLIC PreExecutionCheck
VAR_INPUT
	Check : I_PreExecutionChecks;
END_VAR
Check.IsTrue(ipContainer.IsValid, 'ipContainer must be a valid container');
END_METHOD

END_FUNCTION_BLOCK

// Nodes/Container Statistics/Node_F_VN_MedianElementElementwise_TcVnVector2_USINT
{attribute 'linkalways'} 
{attribute 'no_explicit_call' := 'This FB is a CLASS and must be accessed using methods or properties'}
{attribute 'enable_dynamic_creation'}
FUNCTION_BLOCK Node_F_VN_MedianElementElementwise_TcVnVector2_USINT EXTENDS VisionNode
VAR
    ipContainer : _ITcVnContainer;
    aMedian : _TcVnVector2_USINT;
    hrPrev : _HRESULT(S_OK);
    hresult : _HRESULT(S_OK);
END_VAR

METHOD FB_init : BOOL
VAR_INPUT
	bInitRetains : BOOL; // if TRUE, the retain variables are initialized (warm start / cold start)
	bInCopyCode : BOOL;  // if TRUE, the instance afterwards gets moved into the copy code (online change)
END_VAR
AddInput('ipContainer', ipContainer);
AddInput('aMedian', aMedian);
AddInput('hrPrev', hrPrev);
AddOutput('ipContainer', ipContainer);
AddOutput('hresult',hresult);
END_METHOD

METHOD PUBLIC  Clone : I_Node
VAR
	pNode : POINTER TO Node_F_VN_MedianElementElementwise_TcVnVector2_USINT;
END_VAR
pNode := __NEW(Node_F_VN_MedianElementElementwise_TcVnVector2_USINT);
Clone := pNode^;
END_METHOD

